(* IEC 61131-3 sources: std_i2980_v2.06_cp053/Source/IMM/ieccontrol/MoldGeneral, 17 files *)

(* ---- FBICMProfile.pu ---- *)
(*
/*-------------------------------------------------------------------------
@h    ! WARNING !
@h    The Kemro K2 system (including software) only meets category B according to EN 954-1,
@h    thus it is not intended for usage in safety-relevant control applications in the field
@h    of personal safety (e.g. emergency stop).
@h    To implement potentially necessary safety-relevant control tasks, always use additional
@h    external safety devices that are intended for the particular purpose, and meet the necessary
@h    functional safety.
@h    For further information see EN 954-1 (EN ISO 13849-1) and/or the K2-x00 user manual, chapter
@h    "CE conformity, directives and standards".

- FB build the profile which corresponds to the input values. Acceleration should be sinus curve. The velocity and position will be
  outputed using the intergration (In this FB the lib for integration will be not used).

- In case velocity and acceleration is zero, set value should be set to zero

*)

IMPORT_OVER_LISTFILE
 cApplPlasticsPI
, KAPPL_VisProfile

END_IMPORT

FUNCTION_BLOCK FBICMProfile #DUMMY_EDIT_BLOCK

VAR_INPUT
 ProfileICM : KAPPL_VisProfile (* Profile from visualization with the constant parameters for pos,vel,accl *);
 rTimer : REAL (* Timer for the sin, cos, sin^2 builder *);
 rAcceleration : REAL (* Ramp of velocity *);
 bStart : BOOL (* To start the profile generator *);
 bStop : BOOL (* To stop the profile generator *);
 bTimeModeVisu : BOOL (* Timer mode from the visualization, TRUE:cycle time, FALSE: delay time *);
 rStartPosition : REAL (* Start position *);
END_VAR

VAR_OUTPUT
 bReady : BOOL (* End of profile reached *);
 rSetPos : REAL (* Set Position *);
 rSetVel : REAL (* Set velocity *);
 rSetAcc : REAL (* Set accleration *);
 rSetAccConst : REAL (* Set accleration from visu *);
 rAlgebraSign : REAL (* Direction *);
END_VAR

VAR
 iStage : UDINT (* Stage counter *);
 rPosSumTemp : REAL (* Temp var to count the pos *);
 rCurrStagePos : REAL (* Position of Current stage *);
 iOldStage : UDINT := 0 (* Check if the stage changed *);
 rCurrStageVel : REAL (* Velocity of current stage *);
 rLastStagePos : REAL (* Last stage position  *);
 rPosDiff : REAL (* Absolute position *);
 rCurrStageTime : REAL (* time for current stage(move + delay) *);
 rAcclDecTime : REAL (* Accleration or deceleration time *);
 rMidTime : REAL (* Time for motion with const vel *);
 // rAlgebraSign : REAL (* Algebra sign for direction of motion *);
 rPeriod : REAL (* Periode *);
 rFreq : REAL (* Frequency *);
 rAmpl : REAL (* Amplitude *);
 rCurrAcc : REAL (* Current acceleration *);
 bPosSumAccFinished : BOOL (* If pos summed  *);
 bInited : BOOL (* Flag init *);
 rTimeSumTemp : REAL (* Use to get the actual timer of respect timer *);
 rInternalTimer : REAL (* Internal timer for actual time of actual stage *);
 rTimeStopTemp : REAL (* To get the actual time when stop *);
 bStopInited : BOOL (* Flag of initializing for stop functionality *);
 rCurrVel : REAL (* Current velocity *);
 rAcclDecTimeStop : REAL (* Acc/Deceleration time for stop *);
 rPeriodStop : REAL (* Period for stop *);
 rFreqStop : REAL (* Freq for stop *);
 rAmplStop : REAL (* Amplitude for stop *);
 bStopAcc : BOOL (* Stop during acceleration *);
 bStopConst : BOOL (* Stop during constant movement *);
 rCurrPos : REAL (* Current position *);
 rCalcAccDecTime : REAL (* Calculated acc/dec time to check the time to reach  the vel *);
END_VAR
#BEGIN_EDIT_BLOCK
//********************** Initialize***************************//
IF bStart AND NOT bInited THEN
   //reset generator so it starts at the beginning again
   rCurrAcc := ABS(rAcceleration);
   bReady:= FALSE;
   rPosSumTemp := rStartPosition;
   rTimeSumTemp := 0.0;
   iStage := 1;
   iOldStage := 0;//start with value <> iStage
   // to sum the reached pos at last time
   bPosSumAccFinished := FALSE;
   bInited := TRUE;
   //bStop
   bStopInited := FALSE;
   rTimeStopTemp := 0.0;
   //Flag to check if stop finished in different phase
   bStopAcc:= FALSE;
   bStopConst:= FALSE;

ELSIF NOT bStart THEN
   bInited := FALSE;
   RETURN;
END_IF;

//********************** Calculate and Output ***************************//
IF NOT bReady AND bStart THEN

   //*************************Calculatation*******************************//

   rInternalTimer := rTimer - rTimeSumTemp; //time since start of current stage in s
   rCurrStagePos := ProfileICM.Profile.Points[iStage].rPressure;

   //Get the last position
   IF iStage = 1 THEN
      rLastStagePos := rStartPosition;
   ELSE
      rLastStagePos := ProfileICM.Profile.Points[iStage-1].rPressure;
   END_IF;

   //Get the absolute position
   rPosDiff := ABS(rCurrStagePos - rLastStagePos);
   rCurrStageVel := ABS(ProfileICM.Profile.Points[iStage].rVelocity);

   //avoid singularity
   IF rCurrAcc = 0.0 THEN
      rCurrAcc := 1.0;
   END_IF;
   IF rCurrStageVel = 0.0 THEN
      rCurrStageVel := 1.0;
   END_IF;

   //Check the input values
   //Use the input pos(abs) to calc the acc(dec) time assumming that the profile is triangle without midtime
   //Use this calced time to compare with the input vel.In case that it is smaller that input vel,
   //then we take a new calced vel as the current vel replacing input value
   rCalcAccDecTime := SQRT(rPosDiff/rCurrAcc);
   IF rCurrAcc*rCalcAccDecTime<rCurrStageVel THEN
      rCurrStageVel := rCurrAcc*rCalcAccDecTime;
   END_IF;

   //Get the time between accleration and deccleration
   IF rPosDiff <> 0.0 THEN
      rAcclDecTime := rCurrStageVel/rCurrAcc;
      rMidTime := rPosDiff/rCurrStageVel - rAcclDecTime;
   ELSE
      //The same target position as the last stage is inputed
      //when rPosDiff = 0.0 -> rMidTime = 0 and rAcclDecTime = 0
      rAcclDecTime := 0.0;
      rMidTime := 0.0;
   END_IF;

   //Check the time mode
   IF NOT bTimeModeVisu AND iStage <> iOldStage THEN
      //only standstill time in profile
      rCurrStageTime := ProfileICM.Profile.Points[iStage].rStartPos + rMidTime + 2.0*rAcclDecTime;
      bPosSumAccFinished := FALSE;
      iOldStage := iStage;
   ELSIF bTimeModeVisu AND iStage <> iOldStage THEN
      //time of complete stage in profile
      rCurrStageTime := ProfileICM.Profile.Points[iStage].rStartPos;
      bPosSumAccFinished := FALSE;
      iOldStage := iStage;

      //Error handling to check if enough time
      IF rMidTime + 2.0 * rAcclDecTime > rCurrStageTime THEN
         IF rCurrStageTime <> 0.0 THEN
            rCurrStageTime := rMidTime + 2.0 * rAcclDecTime;
         END_IF;
      END_IF;
   END_IF;

   //****************************Output**********************************//

   //During movement
   IF rInternalTimer < (rMidTime+2.0*rAcclDecTime) AND rInternalTimer < rCurrStageTime THEN
      //(never reached when rPosDiff = 0)
      IF rCurrStagePos - rLastStagePos < 0.0 THEN
         rAlgebraSign := -1.0; //position decreases
      ELSE
         rAlgebraSign := 1.0; //position increases
      END_IF;

      //Frequency,Amplitude,Periode
      rPeriod := 2.0*rAcclDecTime;
      rFreq := 2.0*cApplPlasticsPI/rPeriod;
      rAmpl := 0.5*rCurrStageVel*rFreq;

      //Build the pos,vel,acc
      //pos ~ t+sin(t) only during acceleration or deceleration
      //vel ~ sin˛(t)  only during acceleration or deceleration
      //acc ~ sin(t)   only during acceleration or deceleration

      //acceleration or stop during acceleration
      IF rInternalTimer < rCurrStageVel/rCurrAcc OR bStopAcc THEN
         IF bStop THEN
            //Recalculate parameters for a new deceleration profile if stop during acceleration
            IF NOT bStopInited THEN
               rCurrVel := rSetVel;
               rAcclDecTimeStop := rCurrVel/rCurrAcc;
               rPeriodStop := 2.0*rAcclDecTimeStop;
               rFreqStop := 2.0*cApplPlasticsPI/rPeriodStop;
               rAmplStop := 0.5*rCurrVel*rFreqStop;
               rTimeStopTemp := rInternalTimer;
               rPosSumTemp := rSetPos-rAlgebraSign*rAmplStop*(0.5*rPeriodStop-SIN(rFreqStop*(0.5*rPeriodStop))/rFreqStop)/rFreqStop;
               rCurrPos := rSetPos;
               bStopAcc := TRUE;
               bStopInited := TRUE;
            END_IF;

            //deceleration finished
            IF rInternalTimer >= rTimeStopTemp + rAcclDecTimeStop THEN
               rSetPos := rCurrPos + 0.5*rAcclDecTimeStop*rCurrVel;
               rSetVel := 0.0;
               rSetAccConst := 0.0;
               rSetAcc := 0.0;
               bReady := TRUE;
            ELSE
               //Output a new deceleration profile when stop during acceleration
               rSetPos := rPosSumTemp+rAlgebraSign*rAmplStop*((rInternalTimer-rTimeStopTemp+0.5*rPeriodStop)-SIN(rFreqStop*(rInternalTimer-rTimeStopTemp+0.5*rPeriodStop))/rFreqStop)/rFreqStop;
               rSetVel := 2.0 * rAlgebraSign*rAmplStop*SIN(0.5*rFreqStop*(rInternalTimer-rTimeStopTemp+0.5*rPeriodStop))*SIN(0.5*rFreqStop*(rInternalTimer-rTimeStopTemp+0.5*rPeriodStop))/rFreqStop;
               rSetAccConst := -rAlgebraSign * rCurrAcc;
               rSetAcc := -rAlgebraSign*rAmplStop*SIN(rFreqStop*(rInternalTimer-rTimeStopTemp));
            END_IF;

         ELSE
            //acceleration, no stop and normal movement
            rSetPos := rPosSumTemp+rAlgebraSign*rAmpl*(rInternalTimer-SIN(rFreq*rInternalTimer)/rFreq)/rFreq;
            rSetVel := 2.0 * rAlgebraSign*rAmpl*SIN(0.5*rFreq*rInternalTimer)*SIN(0.5*rFreq*rInternalTimer)/rFreq;
            rSetAccConst :=  rAlgebraSign * rCurrAcc;
            rSetAcc := rAlgebraSign*rAmpl*SIN(rFreq*rInternalTimer);
         END_IF;

      //Movement with const vel or stop during const movement
      ELSIF (rInternalTimer >= rCurrStageVel/rCurrAcc AND rInternalTimer < rCurrStageVel/rCurrAcc+rMidTime) OR bStopConst THEN
         //To build the linear part of the position trajectory, get the initial value only once
         IF NOT bPosSumAccFinished THEN
            rPosSumTemp := rSetPos;
            bPosSumAccFinished := TRUE;
         END_IF;

         IF bStop THEN
            //Just recalculate the mid time when stop during const movement
            IF NOT bStopInited THEN
               rTimeStopTemp := rInternalTimer - rAcclDecTime;
               bStopConst:= TRUE;
               bStopInited := TRUE;
            END_IF;

            //Deceleration finished
            IF rInternalTimer >= rTimeStopTemp + 2.0*rAcclDecTime THEN
               rSetPos := rLastStagePos +  rAlgebraSign * (rAcclDecTime+rTimeStopTemp)*rCurrStageVel;
               rSetVel := 0.0;
               rSetAccConst := 0.0;
               rSetAcc := 0.0;
               bReady := TRUE;
            ELSE
               //deceleration after stop and the deceleration profile not neccessary to be recalculated
               rSetPos := rLastStagePos+rAlgebraSign*rCurrStageVel*rTimeStopTemp+rAlgebraSign*rAmpl*((rInternalTimer-rTimeStopTemp)-SIN(rFreq*(rInternalTimer-rTimeStopTemp))/rFreq)/rFreq;
               rSetVel := 2.0 * rAlgebraSign*rAmpl*SIN(0.5*rFreq*(rInternalTimer-rTimeStopTemp))*SIN(0.5*rFreq*(rInternalTimer-rTimeStopTemp))/rFreq;
               rSetAccConst :=  -rAlgebraSign * rCurrAcc;
               rSetAcc := rAlgebraSign*rAmpl*SIN(rFreq*(rInternalTimer-rTimeStopTemp));
            END_IF;

         ELSE
            //constant movement, no stop and normal movement
            rSetPos := rPosSumTemp + rAlgebraSign*rCurrStageVel*(rInternalTimer-rAcclDecTime);
            rSetVel := rAlgebraSign*rCurrStageVel;
            rSetAccConst := 0.0;
            rSetAcc := 0.0;
         END_IF;
      ELSE
         //deceleration
         //when bStop is set here nothing special happens, we continue our normal stopping
         rSetPos := rLastStagePos+rAlgebraSign*rCurrStageVel*rMidTime+rAlgebraSign*rAmpl*((rInternalTimer-rMidTime)-SIN(rFreq*(rInternalTimer-rMidTime))/rFreq)/rFreq;
         rSetVel := 2.0 * rAlgebraSign*rAmpl*SIN(0.5*rFreq*(rInternalTimer-rMidTime))*SIN(0.5*rFreq*(rInternalTimer-rMidTime))/rFreq;
         rSetAccConst := -rAlgebraSign * rCurrAcc;
         rSetAcc := -rAlgebraSign*rAmpl*SIN(rFreq*(rInternalTimer-rAcclDecTime-rMidTime));
      END_IF;
   ELSIF rInternalTimer >= (rMidTime+2.0*rAcclDecTime) AND rInternalTimer < rCurrStageTime THEN
      //standing still (waiting time)
      rSetPos := rCurrStagePos;
      rSetVel := 0.0;
      rSetAccConst := 0.0;
      rSetAcc := 0.0;
      IF bStop THEN
         bReady := TRUE;
      END_IF;
   ELSE
      rSetPos := rCurrStagePos;
      rSetVel := 0.0;
      rSetAccConst := 0.0;
      rSetAcc := 0.0;
      //end of stage reached
      rPosSumTemp := rCurrStagePos;  //use profile value
      rTimeSumTemp := rTimeSumTemp +  rCurrStageTime;
      IF iStage >= ProfileICM.Profile.iNoOfPoints OR bStop THEN
         //end of profile reached
         bReady := TRUE;
      ELSE
         //end of the stage reached and get the new stage index
         iStage := iStage + 1;
         bPosSumAccFinished := FALSE;
      END_IF;
   END_IF;
END_IF;

;#END_EDIT_BLOCK END_FUNCTION_BLOCK

#END_OF_IEC_PART

@Puma @IecEditor 6 120 @Pou 25
@@@BEG_Comment@@@
/*-------------------------------------------------------------------------
@h    ! WARNING !
@h    The Kemro K2 system (including software) only meets category B according to EN 954-1,
@h    thus it is not intended for usage in safety-relevant control applications in the field
@h    of personal safety (e.g. emergency stop).
@h    To implement potentially necessary safety-relevant control tasks, always use additional
@h    external safety devices that are intended for the particular purpose, and meet the necessary
@h    functional safety.
@h    For further information see EN 954-1 (EN ISO 13849-1) and/or the K2-x00 user manual, chapter
@h    "CE conformity, directives and standards".

- FB build the profile which corresponds to the input values. Acceleration should be sinus curve. The velocity and position will be
  outputed using the intergration (In this FB the lib for integration will be not used).

- In case velocity and acceleration is zero, set value should be set to zero

@@@END_Comment@@@

@BEG_Contents

@BEG_Func
@RT(17)FuncTreeContainer
0
@END_Func

@BEG_Const
@RT(18)ConstTreeContainer
1
@Var @RT(15)cApplPlasticsPI @RT(0) @T @F @DT @RT(4)REAL @RT(0) @T @T @BASIC 0 @F
@F @F
@T
@BEG_Attrib
0 @RT(10)3.14159265 @RT(13)pi=3.14159265
@END_Attrib
1 1 @F @F @F @F

@END_Const

@BEG_Export

@BEG_Kind
@FUNCTION_BLOCK @RT(12)FBICMProfile @STRUCTURED_TEXT
@RT(0) @RT(0) @RT(0)
@END_Kind

@BEG_Dcl
@RT(16)DclTreeContainer
43
@Var @RT(10)ProfileICM @RT(0) @T @T @DERIVED 0 @F @RT(16)KAPPL_VisProfile @F
@T
@BEG_Attrib
3 @RT(0) @RT(72)Profile from visualization with the constant parameters for pos,vel,accl @RT(0)
@END_Attrib
1 1 @F @F @F @F

@Var @RT(6)rTimer @RT(0) @T @F @DT @RT(4)REAL @RT(0) @T @T @BASIC 0 @F
@F @F
@T
@BEG_Attrib
3 @RT(0) @RT(37)Timer for the sin, cos, sin^2 builder @RT(0)
@END_Attrib
1 1 @F @F @F @F

@Var @RT(13)rAcceleration @RT(0) @T @F @DT @RT(4)REAL @RT(0) @T @T @BASIC 0 @F
@F @F
@T
@BEG_Attrib
3 @RT(0) @RT(16)Ramp of velocity @RT(0)
@END_Attrib
1 1 @F @F @F @F

@Var @RT(6)bStart @RT(0) @T @F @DT @RT(4)BOOL @RT(0) @T @T @BASIC 0 @F
@F @F
@T
@BEG_Attrib
3 @RT(0) @RT(30)To start the profile generator @RT(0)
@END_Attrib
1 1 @F @F @F @F

@Var @RT(5)bStop @RT(0) @T @F @DT @RT(4)BOOL @RT(0) @T @T @BASIC 0 @F
@F @F
@T
@BEG_Attrib
3 @RT(0) @RT(29)To stop the profile generator @RT(0)
@END_Attrib
1 1 @F @F @F @F

@Var @RT(13)bTimeModeVisu @RT(0) @T @F @DT @RT(4)BOOL @RT(0) @T @T @BASIC 0 @F
@F @F
@T
@BEG_Attrib
3 @RT(0) @RT(69)Timer mode from the visualization, TRUE:cycle time, FALSE: delay time @RT(0)
@END_Attrib
1 1 @F @F @F @F

@Var @RT(14)rStartPosition @RT(0) @T @F @DT @RT(4)REAL @RT(0) @T @T @BASIC 0 @F
@F @F
@T
@BEG_Attrib
3 @RT(0) @RT(14)Start position @RT(0)
@END_Attrib
1 1 @F @F @F @F

@Var @RT(6)bReady @RT(0) @T @F @DT @RT(4)BOOL @RT(0) @T @T @BASIC 0 @F
@F @F
@T
@BEG_Attrib
3 @RT(0) @RT(22)End of profile reached @RT(0)
@END_Attrib
1 3 @F @F @F @F

@Var @RT(7)rSetPos @RT(0) @T @F @DT @RT(4)REAL @RT(0) @T @T @BASIC 0 @F
@F @F
@T
@BEG_Attrib
3 @RT(0) @RT(12)Set Position @RT(0)
@END_Attrib
1 3 @F @F @F @F

@Var @RT(7)rSetVel @RT(0) @T @F @DT @RT(4)REAL @RT(0) @T @T @BASIC 0 @F
@F @F
@T
@BEG_Attrib
3 @RT(0) @RT(12)Set velocity @RT(0)
@END_Attrib
1 3 @F @F @F @F

@Var @RT(7)rSetAcc @RT(0) @T @F @DT @RT(4)REAL @RT(0) @T @T @BASIC 0 @F
@F @F
@T
@BEG_Attrib
3 @RT(0) @RT(15)Set accleration @RT(0)
@END_Attrib
1 3 @F @F @F @F

@Var @RT(12)rSetAccConst @RT(0) @T @F @DT @RT(4)REAL @RT(0) @T @T @BASIC 0 @F
@F @F
@T
@BEG_Attrib
3 @RT(0) @RT(25)Set accleration from visu @RT(0)
@END_Attrib
1 3 @F @F @F @F

@Var @RT(6)iStage @RT(0) @T @F @DT @RT(5)UDINT @RT(0) @T @T @BASIC 0 @F
@F @F
@T
@BEG_Attrib
3 @RT(0) @RT(13)Stage counter @RT(0)
@END_Attrib
1 0 @F @F @F @F

@Var @RT(11)rPosSumTemp @RT(0) @T @F @DT @RT(4)REAL @RT(0) @T @T @BASIC 0 @F
@F @F
@T
@BEG_Attrib
3 @RT(0) @RT(25)Temp var to count the pos @RT(0)
@END_Attrib
1 0 @F @F @F @F

@Var @RT(13)rCurrStagePos @RT(0) @T @T @RENAMED 0 @T @T @DT @RT(4)REAL @RT(0) @T @T @BASIC 0 @F
@F @F
@T
@BEG_Attrib
3 @RT(0) @RT(25)Position of Current stage @RT(0)
@END_Attrib
1 0 @F @F @F @F

@Var @RT(9)iOldStage @RT(0) @T @F @DT @RT(5)UDINT @RT(0) @T @T @BASIC 0 @F
@F @F
@T
@BEG_Attrib
3 @RT(1)0 @RT(26)Check if the stage changed @RT(0)
@END_Attrib
1 0 @F @F @F @F

@Var @RT(13)rCurrStageVel @RT(0) @T @T @RENAMED 0 @T @T @DT @RT(4)REAL @RT(0) @T @T @BASIC 0 @F
@F @F
@T
@BEG_Attrib
3 @RT(0) @RT(25)Velocity of current stage @RT(0)
@END_Attrib
1 0 @F @F @F @F

@Var @RT(13)rLastStagePos @RT(0) @T @F @DT @RT(4)REAL @RT(0) @T @T @BASIC 0 @F
@F @F
@T
@BEG_Attrib
3 @RT(0) @RT(20)Last stage position  @RT(0)
@END_Attrib
1 0 @F @F @F @F

@Var @RT(8)rPosDiff @RT(0) @T @T @RENAMED 0 @T @T @DT @RT(4)REAL @RT(0) @T @T @BASIC 0 @F
@F @F
@T
@BEG_Attrib
3 @RT(0) @RT(17)Absolute position @RT(0)
@END_Attrib
1 0 @F @F @F @F

@Var @RT(14)rCurrStageTime @RT(0) @T @F @DT @RT(4)REAL @RT(0) @T @T @BASIC 0 @F
@F @F
@T
@BEG_Attrib
3 @RT(0) @RT(36)time for current stage(move + delay) @RT(0)
@END_Attrib
1 0 @F @F @F @F

@Var @RT(12)rAcclDecTime @RT(0) @T @F @DT @RT(4)REAL @RT(0) @T @T @BASIC 0 @F
@F @F
@T
@BEG_Attrib
3 @RT(0) @RT(32)Accleration or deceleration time @RT(0)
@END_Attrib
1 0 @F @F @F @F

@Var @RT(8)rMidTime @RT(0) @T @F @DT @RT(4)REAL @RT(0) @T @T @BASIC 0 @F
@F @F
@T
@BEG_Attrib
3 @RT(0) @RT(30)Time for motion with const vel @RT(0)
@END_Attrib
1 0 @F @F @F @F

@Var @RT(12)rAlgebraSign @RT(0) @T @T @RENAMED 0 @T @T @DT @RT(4)REAL @RT(0) @T @T @BASIC 0 @F
@F @T
@T
@BEG_Attrib
3 @RT(0) @RT(36)Algebra sign for direction of motion @RT(0)
@END_Attrib
1 0 @F @F @F @F

@Var @RT(7)rPeriod @RT(0) @T @T @RENAMED 0 @T @T @DT @RT(4)REAL @RT(0) @T @T @BASIC 0 @F
@F @F
@T
@BEG_Attrib
3 @RT(0) @RT(7)Periode @RT(0)
@END_Attrib
1 0 @F @F @F @F

@Var @RT(5)rFreq @RT(0) @T @T @RENAMED 0 @T @T @DT @RT(4)REAL @RT(0) @T @T @BASIC 0 @F
@F @F
@T
@BEG_Attrib
3 @RT(0) @RT(9)Frequency @RT(0)
@END_Attrib
1 0 @F @F @F @F

@Var @RT(5)rAmpl @RT(0) @T @T @RENAMED 0 @T @T @DT @RT(4)REAL @RT(0) @T @T @BASIC 0 @F
@F @F
@T
@BEG_Attrib
3 @RT(0) @RT(9)Amplitude @RT(0)
@END_Attrib
1 0 @F @F @F @F

@Var @RT(8)rCurrAcc @RT(0) @T @F @DT @RT(4)REAL @RT(0) @T @T @BASIC 0 @F
@F @F
@T
@BEG_Attrib
3 @RT(0) @RT(20)Current acceleration @RT(0)
@END_Attrib
1 0 @F @F @F @F

@Var @RT(18)bPosSumAccFinished @RT(0) @T @F @DT @RT(4)BOOL @RT(0) @T @T @BASIC 0 @F
@F @F
@T
@BEG_Attrib
3 @RT(0) @RT(14)If pos summed  @RT(0)
@END_Attrib
1 0 @F @F @F @F

@Var @RT(7)bInited @RT(0) @T @F @DT @RT(4)BOOL @RT(0) @T @T @BASIC 0 @F
@F @F
@T
@BEG_Attrib
3 @RT(0) @RT(9)Flag init @RT(0)
@END_Attrib
1 0 @F @F @F @F

@Var @RT(12)rTimeSumTemp @RT(0) @T @F @DT @RT(4)REAL @RT(0) @T @T @BASIC 0 @F
@F @F
@T
@BEG_Attrib
3 @RT(0) @RT(44)Use to get the actual timer of respect timer @RT(0)
@END_Attrib
1 0 @F @F @F @F

@Var @RT(14)rInternalTimer @RT(0) @T @F @DT @RT(4)REAL @RT(0) @T @T @BASIC 0 @F
@F @F
@T
@BEG_Attrib
3 @RT(0) @RT(46)Internal timer for actual time of actual stage @RT(0)
@END_Attrib
1 0 @F @F @F @F

@Var @RT(13)rTimeStopTemp @RT(0) @T @F @DT @RT(4)REAL @RT(0) @T @T @BASIC 0 @F
@F @F
@T
@BEG_Attrib
3 @RT(0) @RT(32)To get the actual time when stop @RT(0)
@END_Attrib
1 0 @F @F @F @F

@Var @RT(11)bStopInited @RT(0) @T @F @DT @RT(4)BOOL @RT(0) @T @T @BASIC 0 @F
@F @F
@T
@BEG_Attrib
3 @RT(0) @RT(43)Flag of initializing for stop functionality @RT(0)
@END_Attrib
1 0 @F @F @F @F

@Var @RT(8)rCurrVel @RT(0) @T @F @DT @RT(4)REAL @RT(0) @T @T @BASIC 0 @F
@F @F
@T
@BEG_Attrib
3 @RT(0) @RT(16)Current velocity @RT(0)
@END_Attrib
1 0 @F @F @F @F

@Var @RT(16)rAcclDecTimeStop @RT(0) @T @F @DT @RT(4)REAL @RT(0) @T @T @BASIC 0 @F
@F @F
@T
@BEG_Attrib
3 @RT(0) @RT(30)Acc/Deceleration time for stop @RT(0)
@END_Attrib
1 0 @F @F @F @F

@Var @RT(11)rPeriodStop @RT(0) @T @F @DT @RT(4)REAL @RT(0) @T @T @BASIC 0 @F
@F @F
@T
@BEG_Attrib
3 @RT(0) @RT(15)Period for stop @RT(0)
@END_Attrib
1 0 @F @F @F @F

@Var @RT(9)rFreqStop @RT(0) @T @F @DT @RT(4)REAL @RT(0) @T @T @BASIC 0 @F
@F @F
@T
@BEG_Attrib
3 @RT(0) @RT(13)Freq for stop @RT(0)
@END_Attrib
1 0 @F @F @F @F

@Var @RT(9)rAmplStop @RT(0) @T @F @DT @RT(4)REAL @RT(0) @T @T @BASIC 0 @F
@F @F
@T
@BEG_Attrib
3 @RT(0) @RT(18)Amplitude for stop @RT(0)
@END_Attrib
1 0 @F @F @F @F

@Var @RT(8)bStopAcc @RT(0) @T @F @DT @RT(4)BOOL @RT(0) @T @T @BASIC 0 @F
@F @F
@T
@BEG_Attrib
3 @RT(0) @RT(24)Stop during acceleration @RT(0)
@END_Attrib
1 0 @F @F @F @F

@Var @RT(10)bStopConst @RT(0) @T @F @DT @RT(4)BOOL @RT(0) @T @T @BASIC 0 @F
@F @F
@T
@BEG_Attrib
3 @RT(0) @RT(29)Stop during constant movement @RT(0)
@END_Attrib
1 0 @F @F @F @F

@Var @RT(8)rCurrPos @RT(0) @T @F @DT @RT(4)REAL @RT(0) @T @T @BASIC 0 @F
@F @F
@T
@BEG_Attrib
3 @RT(0) @RT(16)Current position @RT(0)
@END_Attrib
1 0 @F @F @F @F

@Var @RT(15)rCalcAccDecTime @RT(0) @T @F @DT @RT(4)REAL @RT(0) @T @T @BASIC 0 @F
@F @F
@T
@BEG_Attrib
3 @RT(0) @RT(59)Calculated acc/dec time to check the time to reach  the vel @RT(0)
@END_Attrib
1 0 @F @F @F @F

@Var @RT(12)rAlgebraSign @RT(0) @T @F @DT @RT(4)REAL @RT(0) @T @T @BASIC 0 @F
@F @F
@T
@BEG_Attrib
3 @RT(0) @RT(9)Direction @RT(0)
@END_Attrib
1 3 @F @F @F @F

@END_Dcl

@END_Export

@BEG_Body
@TL(227)
//********************** Initialize***************************//
IF bStart AND NOT bInited THEN
   //reset generator so it starts at the beginning again
   rCurrAcc := ABS(rAcceleration);
   bReady:= FALSE;
   rPosSumTemp := rStartPosition;
   rTimeSumTemp := 0.0;
   iStage := 1;
   iOldStage := 0;//start with value <> iStage
   // to sum the reached pos at last time
   bPosSumAccFinished := FALSE;
   bInited := TRUE;
   //bStop
   bStopInited := FALSE;
   rTimeStopTemp := 0.0;
   //Flag to check if stop finished in different phase
   bStopAcc:= FALSE;
   bStopConst:= FALSE;

ELSIF NOT bStart THEN
   bInited := FALSE;
   RETURN;
END_IF;

//********************** Calculate and Output ***************************//
IF NOT bReady AND bStart THEN

   //*************************Calculatation*******************************//

   rInternalTimer := rTimer - rTimeSumTemp; //time since start of current stage in s
   rCurrStagePos := ProfileICM.Profile.Points[iStage].rPressure;

   //Get the last position
   IF iStage = 1 THEN
      rLastStagePos := rStartPosition;
   ELSE
      rLastStagePos := ProfileICM.Profile.Points[iStage-1].rPressure;
   END_IF;

   //Get the absolute position
   rPosDiff := ABS(rCurrStagePos - rLastStagePos);
   rCurrStageVel := ABS(ProfileICM.Profile.Points[iStage].rVelocity);

   //avoid singularity
   IF rCurrAcc = 0.0 THEN
      rCurrAcc := 1.0;
   END_IF;
   IF rCurrStageVel = 0.0 THEN
      rCurrStageVel := 1.0;
   END_IF;

   //Check the input values
   //Use the input pos(abs) to calc the acc(dec) time assumming that the profile is triangle without midtime
   //Use this calced time to compare with the input vel.In case that it is smaller that input vel,
   //then we take a new calced vel as the current vel replacing input value
   rCalcAccDecTime := SQRT(rPosDiff/rCurrAcc);
   IF rCurrAcc*rCalcAccDecTime<rCurrStageVel THEN
      rCurrStageVel := rCurrAcc*rCalcAccDecTime;
   END_IF;

   //Get the time between accleration and deccleration
   IF rPosDiff <> 0.0 THEN
      rAcclDecTime := rCurrStageVel/rCurrAcc;
      rMidTime := rPosDiff/rCurrStageVel - rAcclDecTime;
   ELSE
      //The same target position as the last stage is inputed
      //when rPosDiff = 0.0 -> rMidTime = 0 and rAcclDecTime = 0
      rAcclDecTime := 0.0;
      rMidTime := 0.0;
   END_IF;

   //Check the time mode
   IF NOT bTimeModeVisu AND iStage <> iOldStage THEN
      //only standstill time in profile
      rCurrStageTime := ProfileICM.Profile.Points[iStage].rStartPos + rMidTime + 2.0*rAcclDecTime;
      bPosSumAccFinished := FALSE;
      iOldStage := iStage;
   ELSIF bTimeModeVisu AND iStage <> iOldStage THEN
      //time of complete stage in profile
      rCurrStageTime := ProfileICM.Profile.Points[iStage].rStartPos;
      bPosSumAccFinished := FALSE;
      iOldStage := iStage;

      //Error handling to check if enough time
      IF rMidTime + 2.0 * rAcclDecTime > rCurrStageTime THEN
         IF rCurrStageTime <> 0.0 THEN
            rCurrStageTime := rMidTime + 2.0 * rAcclDecTime;
         END_IF;
      END_IF;
   END_IF;

   //****************************Output**********************************//

   //During movement
   IF rInternalTimer < (rMidTime+2.0*rAcclDecTime) AND rInternalTimer < rCurrStageTime THEN
      //(never reached when rPosDiff = 0)
      IF rCurrStagePos - rLastStagePos < 0.0 THEN
         rAlgebraSign := -1.0; //position decreases
      ELSE
         rAlgebraSign := 1.0; //position increases
      END_IF;

      //Frequency,Amplitude,Periode
      rPeriod := 2.0*rAcclDecTime;
      rFreq := 2.0*cApplPlasticsPI/rPeriod;
      rAmpl := 0.5*rCurrStageVel*rFreq;

      //Build the pos,vel,acc
      //pos ~ t+sin(t) only during acceleration or deceleration
      //vel ~ sin˛(t)  only during acceleration or deceleration
      //acc ~ sin(t)   only during acceleration or deceleration

      //acceleration or stop during acceleration
      IF rInternalTimer < rCurrStageVel/rCurrAcc OR bStopAcc THEN
         IF bStop THEN
            //Recalculate parameters for a new deceleration profile if stop during acceleration
            IF NOT bStopInited THEN
               rCurrVel := rSetVel;
               rAcclDecTimeStop := rCurrVel/rCurrAcc;
               rPeriodStop := 2.0*rAcclDecTimeStop;
               rFreqStop := 2.0*cApplPlasticsPI/rPeriodStop;
               rAmplStop := 0.5*rCurrVel*rFreqStop;
               rTimeStopTemp := rInternalTimer;
               rPosSumTemp := rSetPos-rAlgebraSign*rAmplStop*(0.5*rPeriodStop-SIN(rFreqStop*(0.5*rPeriodStop))/rFreqStop)/rFreqStop;
               rCurrPos := rSetPos;
               bStopAcc := TRUE;
               bStopInited := TRUE;
            END_IF;

            //deceleration finished
            IF rInternalTimer >= rTimeStopTemp + rAcclDecTimeStop THEN
               rSetPos := rCurrPos + 0.5*rAcclDecTimeStop*rCurrVel;
               rSetVel := 0.0;
               rSetAccConst := 0.0;
               rSetAcc := 0.0;
               bReady := TRUE;
            ELSE
               //Output a new deceleration profile when stop during acceleration
               rSetPos := rPosSumTemp+rAlgebraSign*rAmplStop*((rInternalTimer-rTimeStopTemp+0.5*rPeriodStop)-SIN(rFreqStop*(rInternalTimer-rTimeStopTemp+0.5*rPeriodStop))/rFreqStop)/rFreqStop;
               rSetVel := 2.0 * rAlgebraSign*rAmplStop*SIN(0.5*rFreqStop*(rInternalTimer-rTimeStopTemp+0.5*rPeriodStop))*SIN(0.5*rFreqStop*(rInternalTimer-rTimeStopTemp+0.5*rPeriodStop))/rFreqStop;
               rSetAccConst := -rAlgebraSign * rCurrAcc;
               rSetAcc := -rAlgebraSign*rAmplStop*SIN(rFreqStop*(rInternalTimer-rTimeStopTemp));
            END_IF;

         ELSE
            //acceleration, no stop and normal movement
            rSetPos := rPosSumTemp+rAlgebraSign*rAmpl*(rInternalTimer-SIN(rFreq*rInternalTimer)/rFreq)/rFreq;
            rSetVel := 2.0 * rAlgebraSign*rAmpl*SIN(0.5*rFreq*rInternalTimer)*SIN(0.5*rFreq*rInternalTimer)/rFreq;
            rSetAccConst :=  rAlgebraSign * rCurrAcc;
            rSetAcc := rAlgebraSign*rAmpl*SIN(rFreq*rInternalTimer);
         END_IF;

      //Movement with const vel or stop during const movement
      ELSIF (rInternalTimer >= rCurrStageVel/rCurrAcc AND rInternalTimer < rCurrStageVel/rCurrAcc+rMidTime) OR bStopConst THEN
         //To build the linear part of the position trajectory, get the initial value only once
         IF NOT bPosSumAccFinished THEN
            rPosSumTemp := rSetPos;
            bPosSumAccFinished := TRUE;
         END_IF;

         IF bStop THEN
            //Just recalculate the mid time when stop during const movement
            IF NOT bStopInited THEN
               rTimeStopTemp := rInternalTimer - rAcclDecTime;
               bStopConst:= TRUE;
               bStopInited := TRUE;
            END_IF;

            //Deceleration finished
            IF rInternalTimer >= rTimeStopTemp + 2.0*rAcclDecTime THEN
               rSetPos := rLastStagePos +  rAlgebraSign * (rAcclDecTime+rTimeStopTemp)*rCurrStageVel;
               rSetVel := 0.0;
               rSetAccConst := 0.0;
               rSetAcc := 0.0;
               bReady := TRUE;
            ELSE
               //deceleration after stop and the deceleration profile not neccessary to be recalculated
               rSetPos := rLastStagePos+rAlgebraSign*rCurrStageVel*rTimeStopTemp+rAlgebraSign*rAmpl*((rInternalTimer-rTimeStopTemp)-SIN(rFreq*(rInternalTimer-rTimeStopTemp))/rFreq)/rFreq;
               rSetVel := 2.0 * rAlgebraSign*rAmpl*SIN(0.5*rFreq*(rInternalTimer-rTimeStopTemp))*SIN(0.5*rFreq*(rInternalTimer-rTimeStopTemp))/rFreq;
               rSetAccConst :=  -rAlgebraSign * rCurrAcc;
               rSetAcc := rAlgebraSign*rAmpl*SIN(rFreq*(rInternalTimer-rTimeStopTemp));
            END_IF;

         ELSE
            //constant movement, no stop and normal movement
            rSetPos := rPosSumTemp + rAlgebraSign*rCurrStageVel*(rInternalTimer-rAcclDecTime);
            rSetVel := rAlgebraSign*rCurrStageVel;
            rSetAccConst := 0.0;
            rSetAcc := 0.0;
         END_IF;
      ELSE
         //deceleration
         //when bStop is set here nothing special happens, we continue our normal stopping
         rSetPos := rLastStagePos+rAlgebraSign*rCurrStageVel*rMidTime+rAlgebraSign*rAmpl*((rInternalTimer-rMidTime)-SIN(rFreq*(rInternalTimer-rMidTime))/rFreq)/rFreq;
         rSetVel := 2.0 * rAlgebraSign*rAmpl*SIN(0.5*rFreq*(rInternalTimer-rMidTime))*SIN(0.5*rFreq*(rInternalTimer-rMidTime))/rFreq;
         rSetAccConst := -rAlgebraSign * rCurrAcc;
         rSetAcc := -rAlgebraSign*rAmpl*SIN(rFreq*(rInternalTimer-rAcclDecTime-rMidTime));
      END_IF;
   ELSIF rInternalTimer >= (rMidTime+2.0*rAcclDecTime) AND rInternalTimer < rCurrStageTime THEN
      //standing still (waiting time)
      rSetPos := rCurrStagePos;
      rSetVel := 0.0;
      rSetAccConst := 0.0;
      rSetAcc := 0.0;
      IF bStop THEN
         bReady := TRUE;
      END_IF;
   ELSE
      rSetPos := rCurrStagePos;
      rSetVel := 0.0;
      rSetAccConst := 0.0;
      rSetAcc := 0.0;
      //end of stage reached
      rPosSumTemp := rCurrStagePos;  //use profile value
      rTimeSumTemp := rTimeSumTemp +  rCurrStageTime;
      IF iStage >= ProfileICM.Profile.iNoOfPoints OR bStop THEN
         //end of profile reached
         bReady := TRUE;
      ELSE
         //end of the stage reached and get the new stage index
         iStage := iStage + 1;
         bPosSumAccFinished := FALSE;
      END_IF;
   END_IF;
END_IF;

@END_Body

@END_Contents

(* ---- ABAdditionalMoldSafety.pu ---- *)
IMPORT_OVER_LISTFILE
 SET_ALARM
, GET_SYNC_REFTO
, tsDeviceId
, tnOperationMode
, FBLockUnlock
, KSYS_Status

END_IMPORT

ALGORITHM_BLOCK ABAdditionalMoldSafety #DUMMY_EDIT_BLOCK

SYSTEM_VAR
 sv_DeviceId : tsDeviceId (* unique Device Identifier *);
 sv_bMoldOpen : BOOL;
 sv_bMoldClosed : BOOL;
 sv_bInitDone : BOOL;
 sv_bOutputActive : BOOL (* Output is active *);
 sv_OperationMode : tnOperationMode;
 di_MoldOpenProtect : BOOL (* limit switch for mold open maximum position reached *);
 di_MoldCloseProtect : BOOL (* limit switch for mold close minimum position reached *);
 sv_bFALSE : BOOL;
END_VAR

SYSTEM_OBJECT
 erEndPosChangedWithoutMove : ALARM;
 EV_Task_1 : TASK;
 erEndFwdLimitReached : ALARM;
 erEndBwdLimitReached : ALARM;
 PU_Task_7 : TASK;
 TaskMid : TASK;
END_OBJECT

VAR
 mpbHighPresMoldOpenActive : REFTO BOOL;
END_VAR

POSTUPDATE_ALGORITHM pEndPosChanged ON EV_Task_1 WITH sv_bMoldOpen,sv_bMoldClosed

#BEGIN_EDIT_BLOCK
(**************************************** WARNING ********************************************
 *** The KEBA Kemro K2 System including software is not intended for safety control tasks! ***
 ***                       For further information see Comment tab!                        ***
 *********************************************************************************************)

IF NOT sv_bInitDone OR (sv_OperationMode < nHalfAutomatic) THEN
   RETURN;
END_IF;

IF mpbHighPresMoldOpenActive^ THEN
   //On 2 platen IMM´s the mold moves backward during tiebar bwd movement (high pressure mold open - function).
   //In this case a change of mold close endposition is allowed -> no alarm
   RETURN;
END_IF;

IF NOT sv_bOutputActive THEN
    SET_ALARM(Name := erEndPosChangedWithoutMove,
              SubID1 := sv_DeviceId.CompId,
              SubID2 := sv_DeviceId.IndexId);
END_IF;

;#END_EDIT_BLOCK END_ALGORITHM

POSTUPDATE_ALGORITHM pMoldCloseMinLimitSwitch ON PU_Task_7 WITH di_MoldCloseProtect,sv_bInitDone

VAR
 fbLockUnlock : FBLockUnlock;
 bDILinked : BOOL;
 bInit : BOOL := FALSE;
END_VAR
#BEGIN_EDIT_BLOCK
(**************************************** WARNING ********************************************
 *** The KEBA Kemro K2 System including software is not intended for safety control tasks! ***
 ***                       For further information see Comment tab!                        ***
 *********************************************************************************************)

IF NOT sv_bInitDone THEN
   RETURN;
END_IF;

IF NOT bInit THEN
   bDILinked := IS_LINKED(di_MoldCloseProtect);
   fbLockUnlock.DeviceId := sv_DeviceId;
   fbLockUnlock.MoveDir := cMoveFwd;
   fbLockUnlock.MoveId := cMoveAll;
   fbLockUnlock.Alarm.AlarmId := erEndFwdLimitReached;
   fbLockUnlock.bSetAlarmImmediately := TRUE;
   bInit := TRUE;
END_IF;

IF bDILinked THEN

    IF di_MoldCloseProtect THEN
        fbLockUnlock.Mode := nUnlock;
    ELSE
        fbLockUnlock.Mode := nLockAbort;
    END_IF;
    //lock / unlock all fwd movements
    fbLockUnlock();
END_IF;

;#END_EDIT_BLOCK END_ALGORITHM

POSTUPDATE_ALGORITHM pMoldOpenMaxLimitSwitch ON PU_Task_7 WITH di_MoldOpenProtect,sv_bInitDone

VAR
 fbLockUnlock : FBLockUnlock;
 bDILinked : BOOL;
 bInit : BOOL := FALSE;
END_VAR
#BEGIN_EDIT_BLOCK
(**************************************** WARNING ********************************************
 *** The KEBA Kemro K2 System including software is not intended for safety control tasks! ***
 ***                       For further information see Comment tab!                        ***
 *********************************************************************************************)

IF NOT sv_bInitDone THEN
   RETURN;
END_IF;

IF NOT bInit THEN
   bDILinked := IS_LINKED(di_MoldOpenProtect);
   fbLockUnlock.DeviceId := sv_DeviceId;
   fbLockUnlock.MoveDir := cMoveBwd;
   fbLockUnlock.MoveId := cMoveAll;
   fbLockUnlock.Alarm.AlarmId := erEndBwdLimitReached;
   fbLockUnlock.bSetAlarmImmediately := TRUE;
   bInit := TRUE;
END_IF;

IF bDILinked THEN

    IF di_MoldOpenProtect THEN
        fbLockUnlock.Mode := nUnlock;
    ELSE
        fbLockUnlock.Mode := nLockAbort;
    END_IF;
    //lock / unlock all bwd movements
    fbLockUnlock();
END_IF;

;#END_EDIT_BLOCK END_ALGORITHM

PROCESS_ALGORITHM paInit ON TaskMid AUTOSTART

VAR
 s : KSYS_Status;
END_VAR
#BEGIN_EDIT_BLOCK
(**************************************** WARNING ********************************************
 *** The KEBA Kemro K2 System including software is not intended for safety control tasks! ***
 ***                       For further information see Comment tab!                        ***
 *********************************************************************************************)

mpbHighPresMoldOpenActive := GET_SYNC_REFTO('TieBars1.sv_bHighPressureMoldOpenActive', T#0s, s);
IF (s <> KSYS_Status_OK) THEN
   mpbHighPresMoldOpenActive := @sv_bFALSE;
END_IF;

STOP_PROCESS_ALGORITHM();

;#END_EDIT_BLOCK END_ALGORITHM

END_ALGORITHM_BLOCK

#END_OF_IEC_PART

@Puma @IecEditor 6 114 @Pou 25
@@@BEG_Comment@@@

@@@END_Comment@@@

@BEG_Contents

@BEG_Func
@RT(17)FuncTreeContainer
2
@Var @RT(9)SET_ALARM @RT(0) @T @T @DERIVED 0 @F @RT(23)KEBA_STANDARD_PROCEDURE @F
@T
@BEG_Attrib
0 @RT(0) @RT(0)
@END_Attrib
1 1 @F @F @F @F

@Var @RT(14)GET_SYNC_REFTO @RT(0) @T @T @DERIVED 0 @F @RT(34)KEBA_STANDARD_FUNCTION : ANY_REFTO @F
@T
@BEG_Attrib
0 @RT(0) @RT(0)
@END_Attrib
1 1 @F @F @F @F

@END_Func

@BEG_Const
@RT(18)ConstTreeContainer
0
@END_Const

@BEG_Export

@BEG_Kind
@ALGORITHM_BLOCK @RT(22)ABAdditionalMoldSafety @STRUCTURED_TEXT
@RT(0) @RT(0) @RT(0)
@END_Kind

@BEG_Dcl
@RT(16)DclTreeContainer
16
@Var @RT(11)sv_DeviceId @RT(0) @T @T @DERIVED 0 @T @T @DT @RT(10)tsDeviceId @RT(0) @T @T @UNKNOWN 0 @F
@F @F
@T
@BEG_Attrib
3 @RT(0) @RT(24)unique Device Identifier @RT(0)
@END_Attrib
1 8 @F @F @F @F

@Var @RT(12)sv_bMoldOpen @RT(0) @T @F @DT @RT(4)BOOL @RT(0) @T @T @BASIC 0 @F
@F @F
@T
@BEG_Attrib
3 @RT(0) @RT(0) @RT(0)
@END_Attrib
1 8 @F @F @F @F

@Var @RT(14)sv_bMoldClosed @RT(0) @T @F @DT @RT(4)BOOL @RT(0) @T @T @BASIC 0 @F
@F @F
@T
@BEG_Attrib
3 @RT(0) @RT(0) @RT(0)
@END_Attrib
1 8 @F @F @F @F

@Var @RT(12)sv_bInitDone @RT(0) @T @T @RENAMED 0 @T @T @DT @RT(4)BOOL @RT(0) @T @T @BASIC 0 @F
@F @F
@T
@BEG_Attrib
3 @RT(0) @RT(0) @RT(0)
@END_Attrib
1 8 @F @F @F @F

@Var @RT(16)sv_bOutputActive @RT(0) @T @F @DT @RT(4)BOOL @RT(0) @T @T @BASIC 0 @F
@F @F
@T
@BEG_Attrib
3 @RT(0) @RT(16)Output is active @RT(0)
@END_Attrib
1 8 @F @F @F @F

@Var @RT(26)erEndPosChangedWithoutMove @RT(0) @T @F @DT @RT(5)ALARM @RT(0) @T @T @BASIC 0 @F
@F @F
@T
@BEG_Attrib
3 @RT(0) @RT(0) @RT(0)
@END_Attrib
1 7 @F @F @F @F

@Var @RT(9)EV_Task_1 @RT(0) @T @T @RENAMED 0 @T @T @DT @RT(4)TASK @RT(0) @T @T @BASIC 0 @F
@F @F
@T
@BEG_Attrib
3 @RT(0) @RT(0) @RT(0)
@END_Attrib
1 7 @F @F @F @F

@Var @RT(16)sv_OperationMode @RT(0) @T @T @DERIVED 0 @T @T @DT @RT(15)tnOperationMode @RT(0) @T @T @UNKNOWN 0 @F
@F @F
@T
@BEG_Attrib
3 @RT(0) @RT(0) @RT(0)
@END_Attrib
1 8 @F @F @F @F

@Var @RT(18)di_MoldOpenProtect @RT(0) @T @F @DT @RT(4)BOOL @RT(0) @T @T @BASIC 0 @F
@F @F
@T
@BEG_Attrib
3 @RT(0) @RT(51)limit switch for mold open maximum position reached @RT(0)
@END_Attrib
1 8 @F @F @F @F

@Var @RT(19)di_MoldCloseProtect @RT(0) @T @F @DT @RT(4)BOOL @RT(0) @T @T @BASIC 0 @F
@F @F
@T
@BEG_Attrib
3 @RT(0) @RT(52)limit switch for mold close minimum position reached @RT(0)
@END_Attrib
1 8 @F @F @F @F

@Var @RT(20)erEndFwdLimitReached @RT(0) @T @F @DT @RT(5)ALARM @RT(0) @T @T @BASIC 0 @F
@F @F
@T
@BEG_Attrib
3 @RT(0) @RT(0) @RT(0)
@END_Attrib
1 7 @F @F @F @F

@Var @RT(20)erEndBwdLimitReached @RT(0) @T @F @DT @RT(5)ALARM @RT(0) @T @T @BASIC 0 @F
@F @F
@T
@BEG_Attrib
3 @RT(0) @RT(0) @RT(0)
@END_Attrib
1 7 @F @F @F @F

@Var @RT(9)PU_Task_7 @RT(0) @T @F @DT @RT(4)TASK @RT(0) @T @T @BASIC 0 @F
@F @F
@T
@BEG_Attrib
3 @RT(0) @RT(0) @RT(0)
@END_Attrib
1 7 @F @F @F @F

@Var @RT(25)mpbHighPresMoldOpenActive @RT(0) @T @T @REFTO 0 @T @DT @RT(4)BOOL @RT(0) @T @T @BASIC 0 @F
@F @F
@T
@BEG_Attrib
3 @RT(0) @RT(0) @RT(0)
@END_Attrib
1 0 @F @F @F @F

@Var @RT(7)TaskMid @RT(0) @T @T @RENAMED 0 @T @T @DT @RT(4)TASK @RT(0) @T @T @BASIC 0 @F
@F @F
@T
@BEG_Attrib
3 @RT(0) @RT(0) @RT(0)
@END_Attrib
1 7 @F @F @F @F

@Var @RT(9)sv_bFALSE @RT(0) @T @F @DT @RT(4)BOOL @RT(0) @T @T @BASIC 0 @F
@F @F
@T
@BEG_Attrib
3 @RT(0) @RT(0) @RT(0)
@END_Attrib
1 8 @F @F @F @F

@END_Dcl

@END_Export

@BEG_Body

4

@BEG_Export

@BEG_Algo
@POSTUPDATE_ALGORITHM @RT(14)pEndPosChanged @STRUCTURED_TEXT
@RT(0) @RT(27)sv_bMoldOpen,sv_bMoldClosed @RT(9)EV_Task_1 @F @F
@END_Algo

@BEG_Dcl
@RT(16)DclTreeContainer
0
@END_Dcl

@END_Export

@BEG_Export

@BEG_Algo
@POSTUPDATE_ALGORITHM @RT(24)pMoldCloseMinLimitSwitch @STRUCTURED_TEXT
@RT(0) @RT(32)di_MoldCloseProtect,sv_bInitDone @RT(9)PU_Task_7 @F @F
@END_Algo

@BEG_Dcl
@RT(16)DclTreeContainer
3
@Var @RT(12)fbLockUnlock @RT(0) @T @T @DERIVED 0 @T @T @DT @RT(12)FBLockUnlock @RT(0) @T @T @UNKNOWN 0 @F
@F @F
@T
@BEG_Attrib
3 @RT(0) @RT(0) @RT(0)
@END_Attrib
1 0 @F @F @F @F

@Var @RT(9)bDILinked @RT(0) @T @F @DT @RT(4)BOOL @RT(0) @T @T @BASIC 0 @F
@F @F
@T
@BEG_Attrib
3 @RT(0) @RT(0) @RT(0)
@END_Attrib
1 0 @F @F @F @F

@Var @RT(5)bInit @RT(0) @T @F @DT @RT(4)BOOL @RT(0) @T @T @BASIC 0 @F
@F @F
@T
@BEG_Attrib
3 @RT(5)FALSE @RT(0) @RT(0)
@END_Attrib
1 0 @F @F @F @F

@END_Dcl

@END_Export

@BEG_Export

@BEG_Algo
@POSTUPDATE_ALGORITHM @RT(23)pMoldOpenMaxLimitSwitch @STRUCTURED_TEXT
@RT(0) @RT(31)di_MoldOpenProtect,sv_bInitDone @RT(9)PU_Task_7 @F @F
@END_Algo

@BEG_Dcl
@RT(16)DclTreeContainer
3
@Var @RT(12)fbLockUnlock @RT(0) @T @T @DERIVED 0 @T @T @DT @RT(12)FBLockUnlock @RT(0) @T @T @UNKNOWN 0 @F
@F @F
@T
@BEG_Attrib
3 @RT(0) @RT(0) @RT(0)
@END_Attrib
1 0 @F @F @F @F

@Var @RT(9)bDILinked @RT(0) @T @F @DT @RT(4)BOOL @RT(0) @T @T @BASIC 0 @F
@F @F
@T
@BEG_Attrib
3 @RT(0) @RT(0) @RT(0)
@END_Attrib
1 0 @F @F @F @F

@Var @RT(5)bInit @RT(0) @T @F @DT @RT(4)BOOL @RT(0) @T @T @BASIC 0 @F
@F @F
@T
@BEG_Attrib
3 @RT(5)FALSE @RT(0) @RT(0)
@END_Attrib
1 0 @F @F @F @F

@END_Dcl

@END_Export

@BEG_Export

@BEG_Algo
@PROCESS_ALGORITHM @RT(6)paInit @STRUCTURED_TEXT
@RT(0) @RT(0) @RT(7)TaskMid @T @F
@END_Algo

@BEG_Dcl
@RT(16)DclTreeContainer
1
@Var @RT(1)s @RT(0) @T @T @DERIVED 0 @F @RT(11)KSYS_Status @F
@T
@BEG_Attrib
3 @RT(0) @RT(0) @RT(0)
@END_Attrib
1 0 @F @F @F @F

@END_Dcl

@END_Export

@BEG_Body
@TL(21)
(**************************************** WARNING ********************************************
 *** The KEBA Kemro K2 System including software is not intended for safety control tasks! ***
 ***                       For further information see Comment tab!                        ***
 *********************************************************************************************)

IF NOT sv_bInitDone OR (sv_OperationMode < nHalfAutomatic) THEN
   RETURN;
END_IF;

IF mpbHighPresMoldOpenActive^ THEN
   //On 2 platen IMM´s the mold moves backward during tiebar bwd movement (high pressure mold open - function).
   //In this case a change of mold close endposition is allowed -> no alarm
   RETURN;
END_IF;

IF NOT sv_bOutputActive THEN
    SET_ALARM(Name := erEndPosChangedWithoutMove,
              SubID1 := sv_DeviceId.CompId,
              SubID2 := sv_DeviceId.IndexId);
END_IF;

@END_Body

@@@BEG_Comment@@@
@TL(0)

@@@END_Comment@@@

@BEG_Body
@TL(30)
(**************************************** WARNING ********************************************
 *** The KEBA Kemro K2 System including software is not intended for safety control tasks! ***
 ***                       For further information see Comment tab!                        ***
 *********************************************************************************************)

IF NOT sv_bInitDone THEN
   RETURN;
END_IF;

IF NOT bInit THEN
   bDILinked := IS_LINKED(di_MoldCloseProtect);
   fbLockUnlock.DeviceId := sv_DeviceId;
   fbLockUnlock.MoveDir := cMoveFwd;
   fbLockUnlock.MoveId := cMoveAll;
   fbLockUnlock.Alarm.AlarmId := erEndFwdLimitReached;
   fbLockUnlock.bSetAlarmImmediately := TRUE;
   bInit := TRUE;
END_IF;

IF bDILinked THEN

    IF di_MoldCloseProtect THEN
        fbLockUnlock.Mode := nUnlock;
    ELSE
        fbLockUnlock.Mode := nLockAbort;
    END_IF;
    //lock / unlock all fwd movements
    fbLockUnlock();
END_IF;

@END_Body

@@@BEG_Comment@@@
@TL(0)

@@@END_Comment@@@

@BEG_Body
@TL(30)
(**************************************** WARNING ********************************************
 *** The KEBA Kemro K2 System including software is not intended for safety control tasks! ***
 ***                       For further information see Comment tab!                        ***
 *********************************************************************************************)

IF NOT sv_bInitDone THEN
   RETURN;
END_IF;

IF NOT bInit THEN
   bDILinked := IS_LINKED(di_MoldOpenProtect);
   fbLockUnlock.DeviceId := sv_DeviceId;
   fbLockUnlock.MoveDir := cMoveBwd;
   fbLockUnlock.MoveId := cMoveAll;
   fbLockUnlock.Alarm.AlarmId := erEndBwdLimitReached;
   fbLockUnlock.bSetAlarmImmediately := TRUE;
   bInit := TRUE;
END_IF;

IF bDILinked THEN

    IF di_MoldOpenProtect THEN
        fbLockUnlock.Mode := nUnlock;
    ELSE
        fbLockUnlock.Mode := nLockAbort;
    END_IF;
    //lock / unlock all bwd movements
    fbLockUnlock();
END_IF;

@END_Body

@@@BEG_Comment@@@
@TL(0)

@@@END_Comment@@@

@BEG_Body
@TL(12)
(**************************************** WARNING ********************************************
 *** The KEBA Kemro K2 System including software is not intended for safety control tasks! ***
 ***                       For further information see Comment tab!                        ***
 *********************************************************************************************)

mpbHighPresMoldOpenActive := GET_SYNC_REFTO('TieBars1.sv_bHighPressureMoldOpenActive', T#0s, s);
IF (s <> KSYS_Status_OK) THEN
   mpbHighPresMoldOpenActive := @sv_bFALSE;
END_IF;

STOP_PROCESS_ALGORITHM();

@END_Body

@@@BEG_Comment@@@
@TL(0)

@@@END_Comment@@@
@END_Body

@END_Contents

(* ---- ABButtonControl.pu ---- *)
IMPORT_OVER_LISTFILE
 IS_LINKED
, cBarInvert
, cBarRightToLeft
, ABManualButton
, tyPanelButton
, tevPanelButtonRegisterData
, tevPanelButtonRegister
, tsDeviceId
, tsPanelButton

END_IMPORT

ALGORITHM_BLOCK ABButtonControl #DUMMY_EDIT_BLOCK

SYSTEM_VAR
 sv_bTwoButtonOperation : BOOL (* TRUE: two startbuttons are linked; SV is set in OperationMode - FU *);
 sv_bStartButtonsPressed : BOOL (* TRUE: both start buttons are pressed; SV is set in OperationMode - FU *);
 sv_bInitStart : BOOL;
 sv_bMoldOpen : BOOL;
 sv_bMoldClosed : BOOL;
 sv_bDeviceReady : BOOL;
 sv_rMoldStroke : REAL;
 sv_rMoldPosition : REAL;
 sv_iPanelMovementSelector : DINT;
 sv_PanelButtons : tyPanelButton;
 di_ButtonFwd : BOOL;
 di_ButtonBwd : BOOL;
 di_ButtonGeneral1 : BOOL;
 di_ButtonGeneral2 : BOOL;
 sv_bButtonFwd : BOOL;
 sv_bButtonBwd : BOOL;
 sv_DeviceId : tsDeviceId;
END_VAR

SYSTEM_OBJECT
 PU_Task_7 : TASK;
 PU_Task_13 : TASK;
 evPanelButtonRegister : tevPanelButtonRegister;
END_OBJECT

VAR
 abManualButton : ABManualButton;
 evPanelButtonRegisterData : tevPanelButtonRegisterData;
 mpbButtonFwd : REFTO BOOL;
 mpbButtonGeneralFwd : REFTO BOOL;
 mpbButtonGeneralBwd : REFTO BOOL;
 mbDIButtonBwdLinked : BOOL;
 mbDIButtonFwdLinked : BOOL;
 mpiPanelMovementSelector : REFTO DINT;
 mbDIButtonGeneralBwdLinked : BOOL;
 mbDIButtonGeneralFwdLinked : BOOL;
END_VAR

VAR CONSTANT
 cButtonMoveFwdBwd : DINT := 1;
END_VAR

POSTUPDATE_ALGORITHM pRegisterButtons ON PU_Task_13 WITH sv_bInitStart

#BEGIN_EDIT_BLOCK
(**************************************** WARNING ********************************************
 *** The KEBA Kemro K2 System including software is not intended for safety control tasks! ***
 ***                       For further information see Comment tab!                        ***
 *********************************************************************************************)

IF sv_bTwoButtonOperation THEN
   //use two start buttons for starting mold close
   mpbButtonFwd := @sv_bStartButtonsPressed;
ELSE
   //standard case (use panel button)
   mpbButtonFwd := @di_ButtonFwd;
END_IF;

mbDIButtonFwdLinked := IS_LINKED(di_ButtonFwd);
mbDIButtonBwdLinked := IS_LINKED(di_ButtonBwd);

mpbButtonGeneralFwd := EMPTY;
mpbButtonGeneralBwd := EMPTY;

mbDIButtonGeneralFwdLinked := IS_LINKED(di_ButtonGeneral2);
mbDIButtonGeneralBwdLinked := IS_LINKED(di_ButtonGeneral1);

IF (mbDIButtonGeneralFwdLinked AND mbDIButtonGeneralBwdLinked) THEN
    mpiPanelMovementSelector := @sv_iPanelMovementSelector;
END_IF;

// register combined fwd/bwd movement button
evPanelButtonRegisterData.Button.nPanelButtonType := nPanelButtonMovement;
evPanelButtonRegisterData.Button.iCompId := sv_DeviceId.CompId;
evPanelButtonRegisterData.Button.iIndexId := sv_DeviceId.IndexId;
evPanelButtonRegisterData.Button.iButtonId := cButtonMoveFwdBwd;
evPanelButtonRegisterData.Button.pbActionVar1 := @sv_bButtonBwd;
evPanelButtonRegisterData.Button.pbActionVar2 := @sv_bButtonFwd;
evPanelButtonRegisterData.Button.Optional.prActVar := @sv_rMoldPosition;
evPanelButtonRegisterData.Button.Optional.prMaxVar := @sv_rMoldStroke;
evPanelButtonRegisterData.Button.Optional.pbLimitSwitch1 := @sv_bMoldOpen;
evPanelButtonRegisterData.Button.Optional.pbLimitSwitch2 := @sv_bMoldClosed;
evPanelButtonRegisterData.Button.Optional.prMinVar :=  EMPTY;
evPanelButtonRegisterData.Button.Optional.iBarAttr := cBarRightToLeft OR cBarInvert;
SET_EVENT(evPanelButtonRegister, evPanelButtonRegisterData);

;#END_EDIT_BLOCK END_ALGORITHM

POSTUPDATE_ALGORITHM pButtonClose ON PU_Task_7 WITH mpbButtonFwd^,sv_bButtonFwd,mpbButtonGeneralFwd^

VAR
 bButton : BOOL;
END_VAR
#BEGIN_EDIT_BLOCK
(**************************************** WARNING ********************************************
 *** The KEBA Kemro K2 System including software is not intended for safety control tasks! ***
 ***                       For further information see Comment tab!                        ***
 *********************************************************************************************)

// soft panel button
bButton := sv_bButtonFwd;

// hw panel button
IF CHECK_REF(mpbButtonFwd^) THEN
    bButton := bButton OR mpbButtonFwd^;
END_IF;

// external panel button
IF (mbDIButtonGeneralFwdLinked AND CHECK_REF(mpbButtonGeneralFwd^)) THEN
    bButton := bButton OR mpbButtonGeneralFwd^;
END_IF;

abManualButton.aButtonClose(bButtonClose := bButton);

;#END_EDIT_BLOCK END_ALGORITHM

POSTUPDATE_ALGORITHM pButtonOpen ON PU_Task_7 WITH di_ButtonBwd, sv_bButtonBwd,mpbButtonGeneralBwd^

VAR
 bButton : BOOL;
END_VAR
#BEGIN_EDIT_BLOCK
(**************************************** WARNING ********************************************
 *** The KEBA Kemro K2 System including software is not intended for safety control tasks! ***
 ***                       For further information see Comment tab!                        ***
 *********************************************************************************************)

// soft panel button
bButton := sv_bButtonBwd;

// hw panel button
IF mbDIButtonBwdLinked THEN
    bButton := bButton OR di_ButtonBwd;
END_IF;

// external panel button
IF (mbDIButtonGeneralBwdLinked AND CHECK_REF(mpbButtonGeneralBwd^)) THEN
    bButton := bButton OR mpbButtonGeneralBwd^;
END_IF;

abManualButton.aButtonOpen(bButtonOpen := bButton);

;#END_EDIT_BLOCK END_ALGORITHM

POSTUPDATE_ALGORITHM pMoveSelectorChanged ON PU_Task_7 WITH mpiPanelMovementSelector^

VAR
 Button : tsPanelButton;
END_VAR
#BEGIN_EDIT_BLOCK
(**************************************** WARNING ********************************************
 *** The KEBA Kemro K2 System including software is not intended for safety control tasks! ***
 ***                       For further information see Comment tab!                        ***
 *********************************************************************************************)

mpbButtonGeneralFwd := EMPTY;
mpbButtonGeneralBwd := EMPTY;

IF (NOT sv_bDeviceReady) THEN
    // stop active movements
    abManualButton.aButtonClose(bButtonClose := FALSE);
    abManualButton.aButtonOpen(bButtonOpen := FALSE);
END_IF;

IF (sv_iPanelMovementSelector > 0) THEN
    Button := sv_PanelButtons[sv_iPanelMovementSelector];
    IF Button.iCompId = sv_DeviceId.CompId AND
        Button.iIndexId = sv_DeviceId.IndexId THEN
        IF Button.iButtonId = cButtonMoveFwdBwd THEN
            mpbButtonGeneralFwd := @di_ButtonGeneral2;
            mpbButtonGeneralBwd := @di_ButtonGeneral1;
        END_IF;
    END_IF;
END_IF;

;#END_EDIT_BLOCK END_ALGORITHM

END_ALGORITHM_BLOCK

#END_OF_IEC_PART

@Puma @IecEditor 6 150 @Pou 25
@@@BEG_Comment@@@

@@@END_Comment@@@

@BEG_Contents

@BEG_Func
@RT(17)FuncTreeContainer
1
@Var @RT(9)IS_LINKED @RT(0) @T @T @DERIVED 0 @F @RT(22)KEBA_STANDARD_FUNCTION @F
@T
@BEG_Attrib
0 @RT(0) @RT(0)
@END_Attrib
1 1 @F @F @F @F

@END_Func

@BEG_Const
@RT(18)ConstTreeContainer
2
@Var @RT(10)cBarInvert @RT(0) @T @F @DT @RT(4)BYTE @RT(0) @T @T @BASIC 0 @F
@F @F
@T
@BEG_Attrib
0 @RT(1)1 @RT(0)
@END_Attrib
1 1 @F @F @F @F

@Var @RT(15)cBarRightToLeft @RT(0) @T @F @DT @RT(4)BYTE @RT(0) @T @T @BASIC 0 @F
@F @F
@T
@BEG_Attrib
0 @RT(1)2 @RT(0)
@END_Attrib
1 1 @F @F @F @F

@END_Const

@BEG_Export

@BEG_Kind
@ALGORITHM_BLOCK @RT(15)ABButtonControl @STRUCTURED_TEXT
@RT(0) @RT(0) @RT(0)
@END_Kind

@BEG_Dcl
@RT(16)DclTreeContainer
31
@Var @RT(9)PU_Task_7 @RT(0) @T @T @RENAMED 0 @T @T @DT @RT(4)TASK @RT(0) @T @T @BASIC 0 @F
@F @F
@T
@BEG_Attrib
3 @RT(0) @RT(0) @RT(0)
@END_Attrib
1 7 @F @F @F @F

@Var @RT(10)PU_Task_13 @RT(0) @T @T @RENAMED 0 @T @T @DT @RT(4)TASK @RT(0) @T @T @BASIC 0 @F
@F @F
@T
@BEG_Attrib
3 @RT(0) @RT(0) @RT(0)
@END_Attrib
1 7 @F @F @F @F

@Var @RT(14)abManualButton @RT(0) @T @T @DERIVED 0 @T @T @DT @RT(14)ABManualButton @RT(0) @T @T @UNKNOWN 0 @F
@F @F
@T
@BEG_Attrib
3 @RT(0) @RT(0) @RT(0)
@END_Attrib
1 0 @F @F @F @F

@Var @RT(22)sv_bTwoButtonOperation @RT(0) @T @F @DT @RT(4)BOOL @RT(0) @T @T @BASIC 0 @F
@F @F
@T
@BEG_Attrib
3 @RT(0) @RT(66)TRUE: two startbuttons are linked; SV is set in OperationMode - FU @RT(0)
@END_Attrib
1 8 @F @F @F @F

@Var @RT(23)sv_bStartButtonsPressed @RT(0) @T @F @DT @RT(4)BOOL @RT(0) @T @T @BASIC 0 @F
@F @F
@T
@BEG_Attrib
3 @RT(0) @RT(69)TRUE: both start buttons are pressed; SV is set in OperationMode - FU @RT(0)
@END_Attrib
1 8 @F @F @F @F

@Var @RT(13)sv_bInitStart @RT(0) @T @T @RENAMED 0 @T @T @DT @RT(4)BOOL @RT(0) @T @T @BASIC 0 @F
@F @F
@T
@BEG_Attrib
3 @RT(0) @RT(0) @RT(0)
@END_Attrib
1 8 @F @F @F @F

@Var @RT(12)sv_bMoldOpen @RT(0) @T @T @RENAMED 0 @T @T @DT @RT(4)BOOL @RT(0) @T @T @BASIC 0 @F
@F @F
@T
@BEG_Attrib
3 @RT(0) @RT(0) @RT(0)
@END_Attrib
1 8 @F @F @F @F

@Var @RT(14)sv_bMoldClosed @RT(0) @T @T @RENAMED 0 @T @T @DT @RT(4)BOOL @RT(0) @T @T @BASIC 0 @F
@F @F
@T
@BEG_Attrib
3 @RT(0) @RT(0) @RT(0)
@END_Attrib
1 8 @F @F @F @F

@Var @RT(15)sv_bDeviceReady @RT(0) @T @T @RENAMED 0 @T @T @DT @RT(4)BOOL @RT(0) @T @T @BASIC 0 @F
@F @F
@T
@BEG_Attrib
3 @RT(0) @RT(0) @RT(0)
@END_Attrib
1 8 @F @F @F @F

@Var @RT(14)sv_rMoldStroke @RT(0) @T @F @DT @RT(4)REAL @RT(0) @T @T @BASIC 0 @F
@F @F
@T
@BEG_Attrib
3 @RT(0) @RT(0) @RT(0)
@END_Attrib
1 8 @F @F @F @F

@Var @RT(16)sv_rMoldPosition @RT(0) @T @F @DT @RT(4)REAL @RT(0) @T @T @BASIC 0 @F
@F @F
@T
@BEG_Attrib
3 @RT(0) @RT(0) @RT(0)
@END_Attrib
1 8 @F @F @F @F

@Var @RT(25)sv_iPanelMovementSelector @RT(0) @T @F @DT @RT(4)DINT @RT(0) @T @T @BASIC 0 @F
@F @F
@T
@BEG_Attrib
3 @RT(0) @RT(0) @RT(0)
@END_Attrib
1 8 @F @F @F @F

@Var @RT(15)sv_PanelButtons @RT(0) @T @T @DERIVED 0 @T @T @DT @RT(13)tyPanelButton @RT(0) @T @T @UNKNOWN 0 @F
@F @F
@T
@BEG_Attrib
3 @RT(0) @RT(0) @RT(0)
@END_Attrib
1 8 @F @F @F @F

@Var @RT(25)evPanelButtonRegisterData @RT(0) @T @T @DERIVED 0 @T @T @DT @RT(26)tevPanelButtonRegisterData @RT(0) @T @T @UNKNOWN 0 @F
@F @F
@T
@BEG_Attrib
3 @RT(0) @RT(0) @RT(0)
@END_Attrib
1 0 @F @F @F @F

@Var @RT(21)evPanelButtonRegister @RT(0) @T @T @DERIVED 0 @T @T @DT @RT(22)tevPanelButtonRegister @RT(0) @T @T @UNKNOWN 0 @F
@F @F
@T
@BEG_Attrib
3 @RT(0) @RT(0) @RT(0)
@END_Attrib
1 7 @F @F @F @F

@Var @RT(12)di_ButtonFwd @RT(0) @T @T @RENAMED 0 @T @T @DT @RT(4)BOOL @RT(0) @T @T @BASIC 0 @F
@F @F
@T
@BEG_Attrib
3 @RT(0) @RT(0) @RT(0)
@END_Attrib
1 8 @F @F @F @F

@Var @RT(12)di_ButtonBwd @RT(0) @T @T @RENAMED 0 @T @T @DT @RT(4)BOOL @RT(0) @T @T @BASIC 0 @F
@F @F
@T
@BEG_Attrib
3 @RT(0) @RT(0) @RT(0)
@END_Attrib
1 8 @F @F @F @F

@Var @RT(17)di_ButtonGeneral1 @RT(0) @T @F @DT @RT(4)BOOL @RT(0) @T @T @BASIC 0 @F
@F @F
@T
@BEG_Attrib
3 @RT(0) @RT(0) @RT(0)
@END_Attrib
1 8 @F @F @F @F

@Var @RT(17)di_ButtonGeneral2 @RT(0) @T @F @DT @RT(4)BOOL @RT(0) @T @T @BASIC 0 @F
@F @F
@T
@BEG_Attrib
3 @RT(0) @RT(0) @RT(0)
@END_Attrib
1 8 @F @F @F @F

@Var @RT(13)sv_bButtonFwd @RT(0) @T @F @DT @RT(4)BOOL @RT(0) @T @T @BASIC 0 @F
@F @F
@T
@BEG_Attrib
3 @RT(0) @RT(0) @RT(0)
@END_Attrib
1 8 @F @F @F @F

@Var @RT(13)sv_bButtonBwd @RT(0) @T @F @DT @RT(4)BOOL @RT(0) @T @T @BASIC 0 @F
@F @F
@T
@BEG_Attrib
3 @RT(0) @RT(0) @RT(0)
@END_Attrib
1 8 @F @F @F @F

@Var @RT(11)sv_DeviceId @RT(0) @T @T @DERIVED 0 @T @T @DT @RT(10)tsDeviceId @RT(0) @T @T @UNKNOWN 0 @F
@F @F
@T
@BEG_Attrib
3 @RT(0) @RT(0) @RT(0)
@END_Attrib
1 8 @F @F @F @F

@Var @RT(17)cButtonMoveFwdBwd @RT(0) @T @F @DT @RT(4)DINT @RT(0) @T @T @BASIC 0 @F
@F @F
@T
@BEG_Attrib
3 @RT(1)1 @RT(0) @RT(0)
@END_Attrib
1 15 @F @F @F @F

@Var @RT(12)mpbButtonFwd @RT(0) @T @T @REFTO 0 @T @DT @RT(4)BOOL @RT(0) @T @T @BASIC 0 @F
@F @F
@T
@BEG_Attrib
3 @RT(0) @RT(0) @RT(0)
@END_Attrib
1 0 @F @F @F @F

@Var @RT(19)mpbButtonGeneralFwd @RT(0) @T @T @REFTO 0 @T @DT @RT(4)BOOL @RT(0) @T @T @BASIC 0 @F
@F @F
@T
@BEG_Attrib
3 @RT(0) @RT(0) @RT(0)
@END_Attrib
1 0 @F @F @F @F

@Var @RT(19)mpbButtonGeneralBwd @RT(0) @T @T @REFTO 0 @T @DT @RT(4)BOOL @RT(0) @T @T @BASIC 0 @F
@F @F
@T
@BEG_Attrib
3 @RT(0) @RT(0) @RT(0)
@END_Attrib
1 0 @F @F @F @F

@Var @RT(19)mbDIButtonBwdLinked @RT(0) @T @F @DT @RT(4)BOOL @RT(0) @T @T @BASIC 0 @F
@F @F
@T
@BEG_Attrib
3 @RT(0) @RT(0) @RT(0)
@END_Attrib
1 0 @F @F @F @F

@Var @RT(19)mbDIButtonFwdLinked @RT(0) @T @F @DT @RT(4)BOOL @RT(0) @T @T @BASIC 0 @F
@F @F
@T
@BEG_Attrib
3 @RT(0) @RT(0) @RT(0)
@END_Attrib
1 0 @F @F @F @F

@Var @RT(24)mpiPanelMovementSelector @RT(0) @T @T @REFTO 0 @T @DT @RT(4)DINT @RT(0) @T @T @BASIC 0 @F
@F @F
@T
@BEG_Attrib
3 @RT(0) @RT(0) @RT(0)
@END_Attrib
1 0 @F @F @F @F

@Var @RT(26)mbDIButtonGeneralBwdLinked @RT(0) @T @F @DT @RT(4)BOOL @RT(0) @T @T @BASIC 0 @F
@F @F
@T
@BEG_Attrib
3 @RT(0) @RT(0) @RT(0)
@END_Attrib
1 0 @F @F @F @F

@Var @RT(26)mbDIButtonGeneralFwdLinked @RT(0) @T @F @DT @RT(4)BOOL @RT(0) @T @T @BASIC 0 @F
@F @F
@T
@BEG_Attrib
3 @RT(0) @RT(0) @RT(0)
@END_Attrib
1 0 @F @F @F @F

@END_Dcl

@END_Export

@BEG_Body

4

@BEG_Export

@BEG_Algo
@POSTUPDATE_ALGORITHM @RT(16)pRegisterButtons @STRUCTURED_TEXT
@RT(0) @RT(13)sv_bInitStart @RT(10)PU_Task_13 @F @F
@END_Algo

@BEG_Dcl
@RT(16)DclTreeContainer
0
@END_Dcl

@END_Export

@BEG_Export

@BEG_Algo
@POSTUPDATE_ALGORITHM @RT(12)pButtonClose @STRUCTURED_TEXT
@RT(0) @RT(48)mpbButtonFwd^,sv_bButtonFwd,mpbButtonGeneralFwd^ @RT(9)PU_Task_7 @F @F
@END_Algo

@BEG_Dcl
@RT(16)DclTreeContainer
1
@Var @RT(7)bButton @RT(0) @T @F @DT @RT(4)BOOL @RT(0) @T @T @BASIC 0 @F
@F @F
@T
@BEG_Attrib
3 @RT(0) @RT(0) @RT(0)
@END_Attrib
1 0 @F @F @F @F

@END_Dcl

@END_Export

@BEG_Export

@BEG_Algo
@POSTUPDATE_ALGORITHM @RT(11)pButtonOpen @STRUCTURED_TEXT
@RT(0) @RT(48)di_ButtonBwd, sv_bButtonBwd,mpbButtonGeneralBwd^ @RT(9)PU_Task_7 @F @F
@END_Algo

@BEG_Dcl
@RT(16)DclTreeContainer
1
@Var @RT(7)bButton @RT(0) @T @F @DT @RT(4)BOOL @RT(0) @T @T @BASIC 0 @F
@F @F
@T
@BEG_Attrib
3 @RT(0) @RT(0) @RT(0)
@END_Attrib
1 0 @F @F @F @F

@END_Dcl

@END_Export

@BEG_Export

@BEG_Algo
@POSTUPDATE_ALGORITHM @RT(20)pMoveSelectorChanged @STRUCTURED_TEXT
@RT(0) @RT(25)mpiPanelMovementSelector^ @RT(9)PU_Task_7 @F @F
@END_Algo

@BEG_Dcl
@RT(16)DclTreeContainer
1
@Var @RT(6)Button @RT(0) @T @T @DERIVED 0 @T @T @DT @RT(13)tsPanelButton @RT(0) @T @T @UNKNOWN 0 @F
@F @F
@T
@BEG_Attrib
3 @RT(0) @RT(0) @RT(0)
@END_Attrib
1 0 @F @F @F @F

@END_Dcl

@END_Export

@BEG_Body
@TL(42)
(**************************************** WARNING ********************************************
 *** The KEBA Kemro K2 System including software is not intended for safety control tasks! ***
 ***                       For further information see Comment tab!                        ***
 *********************************************************************************************)

IF sv_bTwoButtonOperation THEN
   //use two start buttons for starting mold close
   mpbButtonFwd := @sv_bStartButtonsPressed;
ELSE
   //standard case (use panel button)
   mpbButtonFwd := @di_ButtonFwd;
END_IF;

mbDIButtonFwdLinked := IS_LINKED(di_ButtonFwd);
mbDIButtonBwdLinked := IS_LINKED(di_ButtonBwd);

mpbButtonGeneralFwd := EMPTY;
mpbButtonGeneralBwd := EMPTY;

mbDIButtonGeneralFwdLinked := IS_LINKED(di_ButtonGeneral2);
mbDIButtonGeneralBwdLinked := IS_LINKED(di_ButtonGeneral1);

IF (mbDIButtonGeneralFwdLinked AND mbDIButtonGeneralBwdLinked) THEN
    mpiPanelMovementSelector := @sv_iPanelMovementSelector;
END_IF;

// register combined fwd/bwd movement button
evPanelButtonRegisterData.Button.nPanelButtonType := nPanelButtonMovement;
evPanelButtonRegisterData.Button.iCompId := sv_DeviceId.CompId;
evPanelButtonRegisterData.Button.iIndexId := sv_DeviceId.IndexId;
evPanelButtonRegisterData.Button.iButtonId := cButtonMoveFwdBwd;
evPanelButtonRegisterData.Button.pbActionVar1 := @sv_bButtonBwd;
evPanelButtonRegisterData.Button.pbActionVar2 := @sv_bButtonFwd;
evPanelButtonRegisterData.Button.Optional.prActVar := @sv_rMoldPosition;
evPanelButtonRegisterData.Button.Optional.prMaxVar := @sv_rMoldStroke;
evPanelButtonRegisterData.Button.Optional.pbLimitSwitch1 := @sv_bMoldOpen;
evPanelButtonRegisterData.Button.Optional.pbLimitSwitch2 := @sv_bMoldClosed;
evPanelButtonRegisterData.Button.Optional.prMinVar :=  EMPTY;
evPanelButtonRegisterData.Button.Optional.iBarAttr := cBarRightToLeft OR cBarInvert;
SET_EVENT(evPanelButtonRegister, evPanelButtonRegisterData);

@END_Body

@@@BEG_Comment@@@
@TL(0)

@@@END_Comment@@@

@BEG_Body
@TL(20)
(**************************************** WARNING ********************************************
 *** The KEBA Kemro K2 System including software is not intended for safety control tasks! ***
 ***                       For further information see Comment tab!                        ***
 *********************************************************************************************)

// soft panel button
bButton := sv_bButtonFwd;

// hw panel button
IF CHECK_REF(mpbButtonFwd^) THEN
    bButton := bButton OR mpbButtonFwd^;
END_IF;

// external panel button
IF (mbDIButtonGeneralFwdLinked AND CHECK_REF(mpbButtonGeneralFwd^)) THEN
    bButton := bButton OR mpbButtonGeneralFwd^;
END_IF;

abManualButton.aButtonClose(bButtonClose := bButton);

@END_Body

@@@BEG_Comment@@@
@TL(0)

@@@END_Comment@@@

@BEG_Body
@TL(21)
(**************************************** WARNING ********************************************
 *** The KEBA Kemro K2 System including software is not intended for safety control tasks! ***
 ***                       For further information see Comment tab!                        ***
 *********************************************************************************************)

// soft panel button
bButton := sv_bButtonBwd;

// hw panel button
IF mbDIButtonBwdLinked THEN
    bButton := bButton OR di_ButtonBwd;
END_IF;

// external panel button
IF (mbDIButtonGeneralBwdLinked AND CHECK_REF(mpbButtonGeneralBwd^)) THEN
    bButton := bButton OR mpbButtonGeneralBwd^;
END_IF;

abManualButton.aButtonOpen(bButtonOpen := bButton);

@END_Body

@@@BEG_Comment@@@
@TL(0)

@@@END_Comment@@@

@BEG_Body
@TL(26)
(**************************************** WARNING ********************************************
 *** The KEBA Kemro K2 System including software is not intended for safety control tasks! ***
 ***                       For further information see Comment tab!                        ***
 *********************************************************************************************)

mpbButtonGeneralFwd := EMPTY;
mpbButtonGeneralBwd := EMPTY;

IF (NOT sv_bDeviceReady) THEN
    // stop active movements
    abManualButton.aButtonClose(bButtonClose := FALSE);
    abManualButton.aButtonOpen(bButtonOpen := FALSE);
END_IF;

IF (sv_iPanelMovementSelector > 0) THEN
    Button := sv_PanelButtons[sv_iPanelMovementSelector];
    IF Button.iCompId = sv_DeviceId.CompId AND
        Button.iIndexId = sv_DeviceId.IndexId THEN
        IF Button.iButtonId = cButtonMoveFwdBwd THEN
            mpbButtonGeneralFwd := @di_ButtonGeneral2;
            mpbButtonGeneralBwd := @di_ButtonGeneral1;
        END_IF;
    END_IF;
END_IF;

@END_Body

@@@BEG_Comment@@@
@TL(0)

@@@END_Comment@@@
@END_Body

@END_Contents

(* ---- ABCheckSettings.pu ---- *)
(*
@h    ! WARNING !
@h    The Kemro K2 system (including software) only meets category B according to EN 954-1,
@h    thus it is not intended for usage in safety-relevant control applications in the field
@h    of personal safety (e.g. emergency stop).
@h    To implement potentially necessary safety-relevant control tasks, always use additional
@h    external safety devices that are intended for the particular purpose, and meet the necessary
@h    functional safety.
@h    For further information see EN 954-1 (EN ISO 13849-1) and/or the K2-x00 user manual, chapter
@h    "CE conformity, directives and standards".

AB set the refernces for the endposition monitor blocks.
This refernces denpend on the selected movement mode (position, limit or time)
In time mode the endposition monitoring is also done by this block.
*)

IMPORT_OVER_LISTFILE
 SET_ALARM
, START_PROCESS_ALGORITHM
, STOP_PROCESS_ALGORITHM
, nPositionDependent
, nMoveTimeDependent
, tsEndPosData

END_IMPORT

ALGORITHM_BLOCK ABCheckSettings #DUMMY_EDIT_BLOCK

SYSTEM_VAR
 sv_bInitStart : BOOL;
 sv_MoldFwdMonData : tsEndPosData;
 di_MoldClosed : BOOL;
END_VAR

SYSTEM_OBJECT
 PU_Task_3 : TASK;
END_OBJECT

POSTUPDATE_ALGORITHM pInitSettings ON PU_Task_3 WITH sv_bInitStart

VAR_TEMP
 tmpFwd : tsEndPosData;
END_VAR
#BEGIN_EDIT_BLOCK
(**************************************** WARNING ********************************************
 *** The KEBA Kemro K2 System including software is not intended for safety control tasks! ***
 ***                       For further information see Comment tab!                        ***
 *********************************************************************************************)
tmpFwd := sv_MoldFwdMonData;

IF IS_LINKED (di_MoldClosed)THEN
   tmpFwd.pbDI := @di_MoldClosed;
ELSE
   tmpFwd.pbDI := EMPTY;
END_IF;

// update
sv_MoldFwdMonData := tmpFwd;

;#END_EDIT_BLOCK END_ALGORITHM

END_ALGORITHM_BLOCK

#END_OF_IEC_PART

@Puma @IecEditor 6 103 @Pou 25
@@@BEG_Comment@@@
@h    ! WARNING !
@h    The Kemro K2 system (including software) only meets category B according to EN 954-1,
@h    thus it is not intended for usage in safety-relevant control applications in the field
@h    of personal safety (e.g. emergency stop).
@h    To implement potentially necessary safety-relevant control tasks, always use additional
@h    external safety devices that are intended for the particular purpose, and meet the necessary
@h    functional safety.
@h    For further information see EN 954-1 (EN ISO 13849-1) and/or the K2-x00 user manual, chapter
@h    "CE conformity, directives and standards".

AB set the refernces for the endposition monitor blocks.
This refernces denpend on the selected movement mode (position, limit or time)
In time mode the endposition monitoring is also done by this block.
@@@END_Comment@@@

@BEG_Contents

@BEG_Func
@RT(17)FuncTreeContainer
3
@Var @RT(9)SET_ALARM @RT(0) @T @T @DERIVED 0 @F @RT(23)KEBA_STANDARD_PROCEDURE @F
@T
@BEG_Attrib
0 @RT(0) @RT(0)
@END_Attrib
1 1 @F @F @F @F

@Var @RT(23)START_PROCESS_ALGORITHM @RT(0) @T @T @DERIVED 0 @F @RT(23)KEBA_STANDARD_PROCEDURE @F
@T
@BEG_Attrib
0 @RT(0) @RT(0)
@END_Attrib
1 1 @F @F @F @F

@Var @RT(22)STOP_PROCESS_ALGORITHM @RT(0) @T @T @DERIVED 0 @F @RT(23)KEBA_STANDARD_PROCEDURE @F
@T
@BEG_Attrib
0 @RT(0) @RT(0)
@END_Attrib
1 1 @F @F @F @F

@END_Func

@BEG_Const
@RT(18)ConstTreeContainer
2
@Var @RT(18)nPositionDependent @RT(0) @T @T @DERIVED 0 @F @RT(14)tnMovementMode @F
@T
@BEG_Attrib
0 @RT(1)0 @RT(0)
@END_Attrib
1 1 @F @F @F @F

@Var @RT(18)nMoveTimeDependent @RT(0) @T @T @DERIVED 0 @F @RT(14)tnMovementMode @F
@T
@BEG_Attrib
0 @RT(1)2 @RT(0)
@END_Attrib
1 1 @F @F @F @F

@END_Const

@BEG_Export

@BEG_Kind
@ALGORITHM_BLOCK @RT(15)ABCheckSettings @STRUCTURED_TEXT
@RT(0) @RT(0) @RT(0)
@END_Kind

@BEG_Dcl
@RT(16)DclTreeContainer
4
@Var @RT(13)sv_bInitStart @RT(0) @T @F @DT @RT(4)BOOL @RT(0) @T @T @BASIC 0 @F
@F @F
@T
@BEG_Attrib
3 @RT(0) @RT(0) @RT(0)
@END_Attrib
1 8 @F @F @F @F

@Var @RT(17)sv_MoldFwdMonData @RT(0) @T @T @DERIVED 0 @T @T @DT @RT(12)tsEndPosData @RT(0) @T @T @UNKNOWN 0 @F
@F @F
@T
@BEG_Attrib
3 @RT(0) @RT(0) @RT(0)
@END_Attrib
1 8 @F @F @F @F

@Var @RT(13)di_MoldClosed @RT(0) @T @F @DT @RT(4)BOOL @RT(0) @T @T @BASIC 0 @F
@F @F
@T
@BEG_Attrib
3 @RT(0) @RT(0) @RT(0)
@END_Attrib
1 8 @F @F @F @F

@Var @RT(9)PU_Task_3 @RT(0) @T @F @DT @RT(4)TASK @RT(0) @T @T @BASIC 0 @F
@F @F
@T
@BEG_Attrib
3 @RT(0) @RT(0) @RT(0)
@END_Attrib
1 7 @F @F @F @F

@END_Dcl

@END_Export

@BEG_Body

1

@BEG_Export

@BEG_Algo
@POSTUPDATE_ALGORITHM @RT(13)pInitSettings @STRUCTURED_TEXT
@RT(0) @RT(13)sv_bInitStart @RT(9)PU_Task_3 @F @F
@END_Algo

@BEG_Dcl
@RT(16)DclTreeContainer
1
@Var @RT(6)tmpFwd @RT(0) @T @T @DERIVED 0 @T @T @DT @RT(12)tsEndPosData @RT(0) @T @T @UNKNOWN 0 @F
@F @F
@T
@BEG_Attrib
3 @RT(0) @RT(0) @RT(0)
@END_Attrib
1 4 @F @F @F @F

@END_Dcl

@END_Export

@BEG_Body
@TL(17)
(**************************************** WARNING ********************************************
 *** The KEBA Kemro K2 System including software is not intended for safety control tasks! ***
 ***                       For further information see Comment tab!                        ***
 *********************************************************************************************)
tmpFwd := sv_MoldFwdMonData;

IF IS_LINKED (di_MoldClosed)THEN
   tmpFwd.pbDI := @di_MoldClosed;
ELSE
   tmpFwd.pbDI := EMPTY;
END_IF;

// update
sv_MoldFwdMonData := tmpFwd;

@END_Body

@@@BEG_Comment@@@
@TL(0)

@@@END_Comment@@@
@END_Body

@END_Contents

(* ---- ABDefaultConditions.pu ---- *)
(*
@h    ! WARNING !
@h    The Kemro K2 system (including software) only meets category B according to EN 954-1,
@h    thus it is not intended for usage in safety-relevant control applications in the field
@h    of personal safety (e.g. emergency stop).
@h    To implement potentially necessary safety-relevant control tasks, always use additional
@h    external safety devices that are intended for the particular purpose, and meet the necessary
@h    functional safety.
@h    For further information see EN 954-1 (EN ISO 13849-1) and/or the K2-x00 user manual, chapter
@h    "CE conformity, directives and standards".

This AB monitors following default condition:
If the mold is not open, all ejector fwd movements are locked.

This default condition is not monitored in the following cases:
+ The machine sequence is created by machine sequencer and not by ODC - files
+ "override ejector safety" is activated
+ monitoring is deactivated (sv_bIgnoreDefaultConditions = TRUE)
+ "eject during mold open" is activated
*)

IMPORT_OVER_LISTFILE
 GET_SYNC_REFTO
, cCompEjector
, FBLockUnlock
, KSYS_Status

END_IMPORT

ALGORITHM_BLOCK ABDefaultConditions #DUMMY_EDIT_BLOCK

SYSTEM_VAR
 sv_bMoldOpen : BOOL;
 sv_bOverrideEjectorSafety : BOOL;
 sv_bIgnoreDefaultConditions : BOOL;
 sv_bUseProgramSwitches : BOOL;
 sv_bInitStart : BOOL;
 sv_bInitDone : BOOL;
END_VAR

SYSTEM_OBJECT
 erMoldNotOpen : ALARM;
 PU_Task_7 : TASK;
 PU_Task_3 : TASK;
END_OBJECT

VAR
 mpiNewSequence : REFTO DINT;
 mpbEjectorFwdDuringOpen : REFTO BOOL;
 mpiEjectorSelector : REFTO INT;
END_VAR

ALGORITHM aLockUnlock

VAR
 fbLockUnlock : FBLockUnlock;
END_VAR
#BEGIN_EDIT_BLOCK
(**************************************** WARNING ********************************************
 *** The KEBA Kemro K2 System including software is not intended for safety control tasks! ***
 ***                       For further information see Comment tab!                        ***
 *********************************************************************************************)

IF NOT sv_bInitDone THEN
   RETURN;  //no lock / unlock before sv_bInitDone
END_IF;

IF sv_bIgnoreDefaultConditions OR NOT sv_bUseProgramSwitches THEN
   //sequence programmmed by machine sequencer or
   //default conditions deactivated
   fbLockUnlock.Mode := nUnlock;
ELSE
   //sequence programmed by files and default conditions activated
   //-> check default conditions
   IF sv_bMoldOpen OR mpbEjectorFwdDuringOpen^ THEN
      //mold open or eject during mold open is activated
      fbLockUnlock.Mode := nUnlock;
   ELSE
      fbLockUnlock.Mode := nLockAbort;
   END_IF;
END_IF;

//lock / unlock all ejector fwd movements
//also consider "override ejector safety"
IF sv_bOverrideEjectorSafety THEN
   fbLockUnlock.Mode := nUnlock;
END_IF;

fbLockUnlock.DeviceId.CompId := cCompEjector;
fbLockUnlock.DeviceId.IndexId := 1;
fbLockUnlock.MoveDir := cMoveFwd;
fbLockUnlock.MoveId := cMoveAll;
fbLockUnlock.Alarm.AlarmId := erMoldNotOpen;
fbLockUnlock();

;#END_EDIT_BLOCK END_ALGORITHM

POSTUPDATE_ALGORITHM pInitStart ON PU_Task_7 WITH sv_bInitStart

VAR
 state : KSYS_Status;
END_VAR
#BEGIN_EDIT_BLOCK
(**************************************** WARNING ********************************************
 *** The KEBA Kemro K2 System including software is not intended for safety control tasks! ***
 ***                       For further information see Comment tab!                        ***
 *********************************************************************************************)

//get references
mpiNewSequence := GET_SYNC_REFTO('ODC1.sv_iODCSequenceUpdated', T#0s, state);
mpbEjectorFwdDuringOpen := GET_SYNC_REFTO('CentralCoordination1.sv_bEjectorFwdDuringMldOpen', T#0s, state);
mpiEjectorSelector := GET_SYNC_REFTO('Ejector1.sv_iODCSelector', T#0s, state);

;#END_EDIT_BLOCK END_ALGORITHM

POSTUPDATE_ALGORITHM pCheckDefaultConditions ON PU_Task_3 WITH sv_bMoldOpen,mpiNewSequence^,sv_bIgnoreDefaultConditions,sv_bOverrideEjectorSafety,mpbEjectorFwdDuringOpen^

#BEGIN_EDIT_BLOCK
(**************************************** WARNING ********************************************
 *** The KEBA Kemro K2 System including software is not intended for safety control tasks! ***
 ***                       For further information see Comment tab!                        ***
 *********************************************************************************************)

aLockUnlock();

;#END_EDIT_BLOCK END_ALGORITHM

POSTUPDATE_ALGORITHM pEjectorODCSelector ON PU_Task_7 WITH mpiEjectorSelector^

#BEGIN_EDIT_BLOCK
(**************************************** WARNING ********************************************
 *** The KEBA Kemro K2 System including software is not intended for safety control tasks! ***
 ***                       For further information see Comment tab!                        ***
 *********************************************************************************************)

IF (mpiEjectorSelector^ >= 5) THEN
   //ejector movement after mold close -> deactivate default conditions
   sv_bIgnoreDefaultConditions := TRUE;
ELSE
   sv_bIgnoreDefaultConditions := FALSE;
END_IF;

;#END_EDIT_BLOCK END_ALGORITHM

END_ALGORITHM_BLOCK

#END_OF_IEC_PART

@Puma @IecEditor 6 126 @Pou 25
@@@BEG_Comment@@@
@h    ! WARNING !
@h    The Kemro K2 system (including software) only meets category B according to EN 954-1,
@h    thus it is not intended for usage in safety-relevant control applications in the field
@h    of personal safety (e.g. emergency stop).
@h    To implement potentially necessary safety-relevant control tasks, always use additional
@h    external safety devices that are intended for the particular purpose, and meet the necessary
@h    functional safety.
@h    For further information see EN 954-1 (EN ISO 13849-1) and/or the K2-x00 user manual, chapter
@h    "CE conformity, directives and standards".

This AB monitors following default condition:
If the mold is not open, all ejector fwd movements are locked.

This default condition is not monitored in the following cases:
+ The machine sequence is created by machine sequencer and not by ODC - files
+ "override ejector safety" is activated
+ monitoring is deactivated (sv_bIgnoreDefaultConditions = TRUE)
+ "eject during mold open" is activated
@@@END_Comment@@@

@BEG_Contents

@BEG_Func
@RT(17)FuncTreeContainer
1
@Var @RT(14)GET_SYNC_REFTO @RT(0) @T @T @DERIVED 0 @F @RT(22)KEBA_STANDARD_FUNCTION @F
@T
@BEG_Attrib
0 @RT(0) @RT(0)
@END_Attrib
1 1 @F @F @F @F

@END_Func

@BEG_Const
@RT(18)ConstTreeContainer
1
@Var @RT(12)cCompEjector @RT(0) @T @F @DT @RT(4)DINT @RT(0) @T @T @BASIC 0 @F
@F @F
@T
@BEG_Attrib
0 @RT(3)102 @RT(17)Component Ejector
@END_Attrib
1 1 @F @F @F @F

@END_Const

@BEG_Export

@BEG_Kind
@ALGORITHM_BLOCK @RT(19)ABDefaultConditions @STRUCTURED_TEXT
@RT(0) @RT(0) @RT(0)
@END_Kind

@BEG_Dcl
@RT(16)DclTreeContainer
12
@Var @RT(12)sv_bMoldOpen @RT(0) @T @T @RENAMED 0 @T @T @DT @RT(4)BOOL @RT(0) @T @T @BASIC 0 @F
@F @F
@T
@BEG_Attrib
3 @RT(0) @RT(0) @RT(0)
@END_Attrib
1 8 @F @F @F @F

@Var @RT(14)mpiNewSequence @RT(0) @T @T @REFTO 0 @T @DT @RT(4)DINT @RT(0) @T @T @BASIC 0 @F
@F @F
@T
@BEG_Attrib
3 @RT(0) @RT(0) @RT(0)
@END_Attrib
1 0 @F @F @F @F

@Var @RT(25)sv_bOverrideEjectorSafety @RT(0) @T @T @RENAMED 0 @T @T @DT @RT(4)BOOL @RT(0) @T @T @BASIC 0 @F
@F @F
@T
@BEG_Attrib
3 @RT(0) @RT(0) @RT(0)
@END_Attrib
1 8 @F @F @F @F

@Var @RT(27)sv_bIgnoreDefaultConditions @RT(0) @T @T @RENAMED 0 @T @T @DT @RT(4)BOOL @RT(0) @T @T @BASIC 0 @F
@F @F
@T
@BEG_Attrib
3 @RT(0) @RT(0) @RT(0)
@END_Attrib
1 8 @F @F @F @F

@Var @RT(22)sv_bUseProgramSwitches @RT(0) @T @F @DT @RT(4)BOOL @RT(0) @T @T @BASIC 0 @F
@F @F
@T
@BEG_Attrib
3 @RT(0) @RT(0) @RT(0)
@END_Attrib
1 8 @F @F @F @F

@Var @RT(13)erMoldNotOpen @RT(0) @T @F @DT @RT(5)ALARM @RT(0) @T @T @BASIC 0 @F
@F @F
@T
@BEG_Attrib
3 @RT(0) @RT(0) @RT(0)
@END_Attrib
1 7 @F @F @F @F

@Var @RT(9)PU_Task_7 @RT(0) @T @F @DT @RT(4)TASK @RT(0) @T @T @BASIC 0 @F
@F @F
@T
@BEG_Attrib
3 @RT(0) @RT(0) @RT(0)
@END_Attrib
1 7 @F @F @F @F

@Var @RT(13)sv_bInitStart @RT(0) @T @F @DT @RT(4)BOOL @RT(0) @T @T @BASIC 0 @F
@F @F
@T
@BEG_Attrib
3 @RT(0) @RT(0) @RT(0)
@END_Attrib
1 8 @F @F @F @F

@Var @RT(12)sv_bInitDone @RT(0) @T @F @DT @RT(4)BOOL @RT(0) @T @T @BASIC 0 @F
@F @F
@T
@BEG_Attrib
3 @RT(0) @RT(0) @RT(0)
@END_Attrib
1 8 @F @F @F @F

@Var @RT(23)mpbEjectorFwdDuringOpen @RT(0) @T @T @REFTO 0 @T @DT @RT(4)BOOL @RT(0) @T @T @BASIC 0 @F
@F @F
@T
@BEG_Attrib
3 @RT(0) @RT(0) @RT(0)
@END_Attrib
1 0 @F @F @F @F

@Var @RT(18)mpiEjectorSelector @RT(0) @T @T @REFTO 0 @T @DT @RT(3)INT @RT(0) @T @T @BASIC 0 @F
@F @F
@T
@BEG_Attrib
3 @RT(0) @RT(0) @RT(0)
@END_Attrib
1 0 @F @F @F @F

@Var @RT(9)PU_Task_3 @RT(0) @T @T @RENAMED 0 @T @T @DT @RT(4)TASK @RT(0) @T @T @BASIC 0 @F
@F @F
@T
@BEG_Attrib
3 @RT(0) @RT(0) @RT(0)
@END_Attrib
1 7 @F @F @F @F

@END_Dcl

@END_Export

@BEG_Body

4

@BEG_Export

@BEG_Algo
@ALGORITHM @RT(11)aLockUnlock @STRUCTURED_TEXT
@RT(0) @RT(0) @RT(0) @F @F
@END_Algo

@BEG_Dcl
@RT(16)DclTreeContainer
1
@Var @RT(12)fbLockUnlock @RT(0) @T @T @DERIVED 0 @T @T @DT @RT(12)FBLockUnlock @RT(0) @T @T @UNKNOWN 0 @F
@F @F
@T
@BEG_Attrib
3 @RT(0) @RT(0) @RT(0)
@END_Attrib
1 0 @F @F @F @F

@END_Dcl

@END_Export

@BEG_Export

@BEG_Algo
@POSTUPDATE_ALGORITHM @RT(10)pInitStart @STRUCTURED_TEXT
@RT(0) @RT(13)sv_bInitStart @RT(9)PU_Task_7 @F @F
@END_Algo

@BEG_Dcl
@RT(16)DclTreeContainer
1
@Var @RT(5)state @RT(0) @T @T @DERIVED 0 @T @T @DT @RT(11)KSYS_Status @RT(0) @T @T @UNKNOWN 0 @F
@F @F
@T
@BEG_Attrib
3 @RT(0) @RT(0) @RT(0)
@END_Attrib
1 0 @F @F @F @F

@END_Dcl

@END_Export

@BEG_Export

@BEG_Algo
@POSTUPDATE_ALGORITHM @RT(23)pCheckDefaultConditions @STRUCTURED_TEXT
@RT(0) @RT(107)sv_bMoldOpen,mpiNewSequence^,sv_bIgnoreDefaultConditions,sv_bOverrideEjectorSafety,mpbEjectorFwdDuringOpen^ @RT(9)PU_Task_3 @F @F
@END_Algo

@BEG_Dcl
@RT(16)DclTreeContainer
0
@END_Dcl

@END_Export

@BEG_Export

@BEG_Algo
@POSTUPDATE_ALGORITHM @RT(19)pEjectorODCSelector @STRUCTURED_TEXT
@RT(0) @RT(19)mpiEjectorSelector^ @RT(9)PU_Task_7 @F @F
@END_Algo

@BEG_Dcl
@RT(16)DclTreeContainer
0
@END_Dcl

@END_Export

@BEG_Body
@TL(40)
(**************************************** WARNING ********************************************
 *** The KEBA Kemro K2 System including software is not intended for safety control tasks! ***
 ***                       For further information see Comment tab!                        ***
 *********************************************************************************************)

IF NOT sv_bInitDone THEN
   RETURN;  //no lock / unlock before sv_bInitDone
END_IF;

IF sv_bIgnoreDefaultConditions OR NOT sv_bUseProgramSwitches THEN
   //sequence programmmed by machine sequencer or
   //default conditions deactivated
   fbLockUnlock.Mode := nUnlock;
ELSE
   //sequence programmed by files and default conditions activated
   //-> check default conditions
   IF sv_bMoldOpen OR mpbEjectorFwdDuringOpen^ THEN
      //mold open or eject during mold open is activated
      fbLockUnlock.Mode := nUnlock;
   ELSE
      fbLockUnlock.Mode := nLockAbort;
   END_IF;
END_IF;

//lock / unlock all ejector fwd movements
//also consider "override ejector safety"
IF sv_bOverrideEjectorSafety THEN
   fbLockUnlock.Mode := nUnlock;
END_IF;

fbLockUnlock.DeviceId.CompId := cCompEjector;
fbLockUnlock.DeviceId.IndexId := 1;
fbLockUnlock.MoveDir := cMoveFwd;
fbLockUnlock.MoveId := cMoveAll;
fbLockUnlock.Alarm.AlarmId := erMoldNotOpen;
fbLockUnlock();

@END_Body

@@@BEG_Comment@@@
@TL(0)

@@@END_Comment@@@

@BEG_Body
@TL(10)
(**************************************** WARNING ********************************************
 *** The KEBA Kemro K2 System including software is not intended for safety control tasks! ***
 ***                       For further information see Comment tab!                        ***
 *********************************************************************************************)

//get references
mpiNewSequence := GET_SYNC_REFTO('ODC1.sv_iODCSequenceUpdated', T#0s, state);
mpbEjectorFwdDuringOpen := GET_SYNC_REFTO('CentralCoordination1.sv_bEjectorFwdDuringMldOpen', T#0s, state);
mpiEjectorSelector := GET_SYNC_REFTO('Ejector1.sv_iODCSelector', T#0s, state);

@END_Body

@@@BEG_Comment@@@
@TL(0)

@@@END_Comment@@@

@BEG_Body
@TL(7)
(**************************************** WARNING ********************************************
 *** The KEBA Kemro K2 System including software is not intended for safety control tasks! ***
 ***                       For further information see Comment tab!                        ***
 *********************************************************************************************)

aLockUnlock();

@END_Body

@@@BEG_Comment@@@
@TL(0)

@@@END_Comment@@@

@BEG_Body
@TL(12)
(**************************************** WARNING ********************************************
 *** The KEBA Kemro K2 System including software is not intended for safety control tasks! ***
 ***                       For further information see Comment tab!                        ***
 *********************************************************************************************)

IF (mpiEjectorSelector^ >= 5) THEN
   //ejector movement after mold close -> deactivate default conditions
   sv_bIgnoreDefaultConditions := TRUE;
ELSE
   sv_bIgnoreDefaultConditions := FALSE;
END_IF;

@END_Body

@@@BEG_Comment@@@
@TL(0)

@@@END_Comment@@@
@END_Body

@END_Contents
